LIN {X 0,Y 286.742,Z 491.523,A -85,B 0,C 180,E1 -18513.428,E2 -18513.428} C_VEL
LIN {X 0,Y 283.186,Z 502.115,A -85,B 0,C 180,E1 -18515.045,E2 -18515.045} C_VEL
LIN {X 0,Y 279.87,Z 510.827,A -85,B 0,C 180,E1 -18516.702,E2 -18516.702} C_VEL
LIN {X 0,Y 276.057,Z 519.397,A -85,B 0,C 180,E1 -18518.728,E2 -18518.728} C_VEL
LIN {X 0,Y 272.636,Z 526.32,A -85,B 0,C 180,E1 -18520.811,E2 -18520.811} C_VEL
LIN {X 0,Y 269.962,Z 531.061,A -85,B 0,C 180,E1 -18522.579,E2 -18522.579} C_VEL
LIN {X 0,Y 267.064,Z 535.632,A -85,B 0,C 180,E1 -18524.742,E2 -18524.742} C_VEL
LIN {X 0,Y 265.332,Z 538.078,A -85,B 0,C 180,E1 -18526.208,E2 -18526.208} C_VEL
LIN {X 0,Y 263.694,Z 540.035,A -85,B 0,C 180,E1 -18527.688,E2 -18527.688} C_VEL
LIN {X 0,Y 262.269,Z 541.552,A -85,B 0,C 180,E1 -18529.188,E2 -18529.188} C_VEL
LIN {X 0,Y 260.929,Z 542.67,A -85,B 0,C 180,E1 -18530.699,E2 -18530.699} C_VEL
LIN {X 0,Y 259.796,Z 543.334,A -85,B 0,C 180,E1 -18532.226,E2 -18532.226} C_VEL
LIN {X 0,Y 257.917,Z 543.43,A -85,B 0,C 180,E1 -18535.31,E2 -18535.31} C_VEL
LIN {X 0,Y 257.232,Z 542.868,A -85,B 0,C 180,E1 -18536.867,E2 -18536.867} C_VEL
LIN {X 0,Y 256.673,Z 541.852,A -85,B 0,C 180,E1 -18538.43,E2 -18538.43} C_VEL
LIN {X 0,Y 256.227,Z 540.428,A -85,B 0,C 180,E1 -18539.999,E2 -18539.999} C_VEL
LIN {X 0,Y 255.594,Z 537.491,A -85,B 0,C 180,E1 -18542.363,E2 -18542.363} C_VEL
LIN {X 0,Y 255.538,Z 533.499,A -85,B 0,C 180,E1 -18544.732,E2 -18544.732} C_VEL
LIN {X 0,Y 255.707,Z 527.917,A -85,B 0,C 180,E1 -18547.289,E2 -18547.289} C_VEL
LIN {X 0,Y 256.033,Z 520.721,A -85,B 0,C 180,E1 -18549.878,E2 -18549.878} C_VEL
LIN {X 0,Y 256.482,Z 512.466,A -85,B 0,C 180,E1 -18552.26,E2 -18552.26} C_VEL
LIN {X 0,Y 257.064,Z 504.113,A -85,B 0,C 180,E1 -18554.243,E2 -18554.243} C_VEL
LIN {X 0,Y 257.823,Z 493.991,A -85,B 0,C 180,E1 -18556.224,E2 -18556.224} C_VEL
LIN {X 0,Y 258.627,Z 482.98,A -85,B 0,C 180,E1 -18557.991,E2 -18557.991} C_VEL
LIN {X 0,Y 259.558,Z 470.695,A -85,B 0,C 180,E1 -18559.576,E2 -18559.576} C_VEL
LIN {X 0,Y 260.256,Z 456.947,A -85,B 0,C 180,E1 -18560.965,E2 -18560.965} C_VEL
LIN {X 0,Y 260.958,Z 443.101,A -85,B 0,C 180,E1 -18561.994,E2 -18561.994} C_VEL
LIN {X 0,Y 261.321,Z 428.706,A -85,B 0,C 180,E1 -18562.742,E2 -18562.742} C_VEL
LIN {X 0,Y 263.063,Z 376.798,A -85,B 0,C 180,E1 -18564.915,E2 -18564.915} C_VEL
LIN {X 0,Y 263.115,Z 373.058,A -85,B 0,C 180,E1 -18565.074,E2 -18565.074} C_VEL
LIN {X 0,Y 256.217,Z 349.569,A -85,B 0,C 180,E1 -18566.43,E2 -18566.43} C_VEL
LIN {X 0,Y 256.113,Z 349.578,A -85,B 0,C 180,E1 -18569.599,E2 -18569.599} C_VEL
LIN {X 0,Y 256.067,Z 349.587,A -85,B 0,C 180,E1 -18573.292,E2 -18573.292} C_VEL
LIN {X 0,Y 256.112,Z 349.58,A -85,B 0,C 180,E1 -18577.27,E2 -18577.27} C_VEL
LIN {X 0,Y 256.053,Z 349.589,A -85,B 0,C 180,E1 -18581.203,E2 -18581.203} C_VEL
LIN {X 0,Y 256.06,Z 349.586,A -85,B 0,C 180,E1 -18585.529,E2 -18585.529} C_VEL
LIN {X 0,Y 256.055,Z 349.591,A -85,B 0,C 180,E1 -18588.797,E2 -18588.797} C_VEL
LIN {X 0,Y 256.143,Z 349.579,A -85,B 0,C 180,E1 -18592.87,E2 -18592.87} C_VEL
LIN {X 0,Y 256.082,Z 349.587,A -85,B 0,C 180,E1 -18596.709,E2 -18596.709} C_VEL
LIN {X 0,Y 256.124,Z 349.579,A -85,B 0,C 180,E1 -18601.409,E2 -18601.409} C_VEL
LIN {X 0,Y 256.164,Z 349.573,A -85,B 0,C 180,E1 -18605.699,E2 -18605.699} C_VEL
LIN {X 0,Y 256.165,Z 349.574,A -85,B 0,C 180,E1 -18609.105,E2 -18609.105} C_VEL
LIN {X 0,Y 256.297,Z 349.557,A -85,B 0,C 180,E1 -18614.085,E2 -18614.085} C_VEL
LIN {X 0,Y 256.307,Z 349.556,A -85,B 0,C 180,E1 -18618.934,E2 -18618.934} C_VEL
LIN {X 0,Y 256.538,Z 349.527,A -85,B 0,C 180,E1 -18622.127,E2 -18622.127} C_VEL
LIN {X 0,Y 256.712,Z 349.508,A -85,B 0,C 180,E1 -18628.431,E2 -18628.431} C_VEL
LIN {X 0,Y 256.712,Z 349.505,A -85,B 0,C 180,E1 -18631.569,E2 -18631.569} C_VEL
LIN {X 0,Y 256.538,Z 349.527,A -85,B 0,C 180,E1 -18637.873,E2 -18637.873} C_VEL
LIN {X 0,Y 256.307,Z 349.556,A -85,B 0,C 180,E1 -18641.066,E2 -18641.066} C_VEL
LIN {X 0,Y 256.298,Z 349.558,A -85,B 0,C 180,E1 -18645.915,E2 -18645.915} C_VEL
LIN {X 0,Y 256.165,Z 349.574,A -85,B 0,C 180,E1 -18650.896,E2 -18650.896} C_VEL
LIN {X 0,Y 256.187,Z 349.569,A -85,B 0,C 180,E1 -18655.139,E2 -18655.139} C_VEL
LIN {X 0,Y 256.102,Z 349.582,A -85,B 0,C 180,E1 -18659.602,E2 -18659.602} C_VEL
LIN {X 0,Y 256.084,Z 349.582,A -85,B 0,C 180,E1 -18663.291,E2 -18663.291} C_VEL
LIN {X 0,Y 256.127,Z 349.578,A -85,B 0,C 180,E1 -18667.276,E2 -18667.276} C_VEL
LIN {X 0,Y 256.056,Z 349.586,A -85,B 0,C 180,E1 -18671.204,E2 -18671.204} C_VEL
LIN {X 0,Y 256.057,Z 349.588,A -85,B 0,C 180,E1 -18675.531,E2 -18675.531} C_VEL
LIN {X 0,Y 256.054,Z 349.587,A -85,B 0,C 180,E1 -18678.798,E2 -18678.798} C_VEL
LIN {X 0,Y 256.139,Z 349.576,A -85,B 0,C 180,E1 -18682.87,E2 -18682.87} C_VEL
LIN {X 0,Y 256.132,Z 349.577,A -85,B 0,C 180,E1 -18687.122,E2 -18687.122} C_VEL
LIN {X 0,Y 263.843,Z 373.942,A -85,B 0,C 180,E1 -18688.527,E2 -18688.527} C_VEL
LIN {X 0,Y 261.875,Z 433.631,A -85,B 0,C 180,E1 -18690.895,E2 -18690.895} C_VEL
LIN {X 0,Y 261.396,Z 447.781,A -85,B 0,C 180,E1 -18691.715,E2 -18691.715} C_VEL
LIN {X 0,Y 260.706,Z 461.252,A -85,B 0,C 180,E1 -18692.824,E2 -18692.824} C_VEL
LIN {X 0,Y 259.893,Z 473.611,A -85,B 0,C 180,E1 -18694.149,E2 -18694.149} C_VEL
LIN {X 0,Y 258.984,Z 485.469,A -85,B 0,C 180,E1 -18695.768,E2 -18695.768} C_VEL
LIN {X 0,Y 258.047,Z 496.288,A -85,B 0,C 180,E1 -18697.587,E2 -18697.587} C_VEL
LIN {X 0,Y 257.243,Z 506.028,A -85,B 0,C 180,E1 -18699.615,E2 -18699.615} C_VEL
LIN {X 0,Y 256.505,Z 515.525,A -85,B 0,C 180,E1 -18702.048,E2 -18702.048} C_VEL
LIN {X 0,Y 255.992,Z 523.081,A -85,B 0,C 180,E1 -18704.475,E2 -18704.475} C_VEL
LIN {X 0,Y 255.613,Z 530.03,A -85,B 0,C 180,E1 -18707.294,E2 -18707.294} C_VEL
LIN {X 0,Y 255.63,Z 534.568,A -85,B 0,C 180,E1 -18709.707,E2 -18709.707} C_VEL
LIN {X 0,Y 255.9,Z 537.977,A -85,B 0,C 180,E1 -18712.108,E2 -18712.108} C_VEL
LIN {X 0,Y 256.113,Z 539.674,A -85,B 0,C 180,E1 -18713.699,E2 -18713.699} C_VEL
LIN {X 0,Y 256.404,Z 540.938,A -85,B 0,C 180,E1 -18715.284,E2 -18715.284} C_VEL
LIN {X 0,Y 256.951,Z 541.725,A -85,B 0,C 180,E1 -18716.865,E2 -18716.865} C_VEL
LIN {X 0,Y 257.624,Z 542.11,A -85,B 0,C 180,E1 -18718.438,E2 -18718.438} C_VEL
LIN {X 0,Y 258.435,Z 542.082,A -85,B 0,C 180,E1 -18720.001,E2 -18720.001} C_VEL
LIN {X 0,Y 259.323,Z 541.593,A -85,B 0,C 180,E1 -18721.554,E2 -18721.554} C_VEL
LIN {X 0,Y 261.561,Z 539.402,A -85,B 0,C 180,E1 -18724.624,E2 -18724.624} C_VEL
LIN {X 0,Y 263.689,Z 536.578,A -85,B 0,C 180,E1 -18726.889,E2 -18726.889} C_VEL
LIN {X 0,Y 266.034,Z 532.7,A -85,B 0,C 180,E1 -18729.121,E2 -18729.121} C_VEL
LIN {X 0,Y 267.361,Z 530.257,A -85,B 0,C 180,E1 -18730.227,E2 -18730.227} C_VEL
LIN {X 0,Y 268.185,Z 527.805,A -85,B 0,C 180,E1 -18731.362,E2 -18731.362} C_VEL
LIN {X 0,Y 268.143,Z 523.856,A -85,B 0,C 180,E1 -18733.306,E2 -18733.306} C_VEL
LIN {X 0,Y 268.21,Z 519.378,A -85,B 0,C 180,E1 -18735.187,E2 -18735.187} C_VEL
LIN {X 0,Y 269.162,Z 516.063,A -85,B 0,C 180,E1 -18736.204,E2 -18736.204} C_VEL
LIN {X 0,Y 272.495,Z 507.969,A -85,B 0,C 180,E1 -18738.03,E2 -18738.03} C_VEL
LIN {X 0,Y 275.746,Z 498.639,A -85,B 0,C 180,E1 -18739.738,E2 -18739.738} C_VEL
LIN {X 0,Y 279.246,Z 487.143,A -85,B 0,C 180,E1 -18741.405,E2 -18741.405} C_VEL
LIN {X 0,Y 282.117,Z 475.634,A -85,B 0,C 180,E1 -18742.715,E2 -18742.715} C_VEL
LIN {X 0,Y 284.548,Z 462.972,A -85,B 0,C 180,E1 -18743.857,E2 -18743.857} C_VEL
LIN {X 0,Y 286.529,Z 448.771,A -85,B 0,C 180,E1 -18744.817,E2 -18744.817} C_VEL
LIN {X 0,Y 289.784,Z 421.766,A -85,B 0,C 180,E1 -18746.079,E2 -18746.079} C_VEL
LIN {X 0,Y 291.826,Z 407.158,A -85,B 0,C 180,E1 -18746.682,E2 -18746.682} C_VEL
LIN {X 0,Y 288.803,Z 401.044,A -85,B 0,C 180,E1 -18748.509,E2 -18748.509} C_VEL
LIN {X 0,Y 286.95,Z 397.572,A -85,B 0,C 180,E1 -18749.809,E2 -18749.809} C_VEL
LIN {X 0,Y 285.256,Z 394.534,A -85,B 0,C 180,E1 -18751.158,E2 -18751.158} C_VEL
LIN {X 0,Y 283.356,Z 391.067,A -85,B 0,C 180,E1 -18753.009,E2 -18753.009} C_VEL
LIN {X 0,Y 281.225,Z 387.965,A -85,B 0,C 180,E1 -18755.844,E2 -18755.844} C_VEL
LIN {X 0,Y 280.356,Z 386.885,A -85,B 0,C 180,E1 -18757.914,E2 -18757.914} C_VEL
LIN {X 0,Y 279.977,Z 387.1,A -85,B 0,C 180,E1 -18760.122,E2 -18760.122} C_VEL
LIN {X 0,Y 280.903,Z 389.538,A -85,B 0,C 180,E1 -18763.905,E2 -18763.905} C_VEL
LIN {X 0,Y 281.598,Z 390.488,A -85,B 0,C 180,E1 -18764.946,E2 -18764.946} C_VEL
LIN {X 0,Y 284.076,Z 395.271,A -85,B 0,C 180,E1 -18767.92,E2 -18767.92} C_VEL
LIN {X 0,Y 285.9,Z 398.582,A -85,B 0,C 180,E1 -18769.468,E2 -18769.468} C_VEL
LIN {X 0,Y 287.386,Z 407.637,A -85,B 0,C 180,E1 -18771.281,E2 -18771.281} C_VEL
LIN {X 0,Y 287.167,Z 422.972,A -85,B 0,C 180,E1 -18772.78,E2 -18772.78} C_VEL
LIN {X 0,Y 286.547,Z 444.861,A -85,B 0,C 180,E1 -18774.577,E2 -18774.577} C_VEL
LIN {X 0,Y 285.739,Z 460.739,A -85,B 0,C 180,E1 -18775.664,E2 -18775.664} C_VEL
LIN {X 0,Y 281.973,Z 489.26,A -85,B 0,C 180,E1 -18776.906,E2 -18776.906} C_VEL
LIN {X 0,Y 279.037,Z 503.696,A -85,B 0,C 180,E1 -18777.748,E2 -18777.748} C_VEL
LIN {X 0,Y 275.393,Z 517.912,A -85,B 0,C 180,E1 -18778.883,E2 -18778.883} C_VEL
LIN {X 0,Y 271.17,Z 531.452,A -85,B 0,C 180,E1 -18780.286,E2 -18780.286} C_VEL
LIN {X 0,Y 266.886,Z 543.474,A -85,B 0,C 180,E1 -18781.919,E2 -18781.919} C_VEL
LIN {X 0,Y 262.716,Z 554.359,A -85,B 0,C 180,E1 -18783.807,E2 -18783.807} C_VEL
LIN {X 0,Y 258.893,Z 564.083,A -85,B 0,C 180,E1 -18785.971,E2 -18785.971} C_VEL
LIN {X 0,Y 254.961,Z 573.385,A -85,B 0,C 180,E1 -18788.577,E2 -18788.577} C_VEL
LIN {X 0,Y 252.27,Z 579.962,A -85,B 0,C 180,E1 -18790.934,E2 -18790.934} C_VEL
LIN {X 0,Y 250.077,Z 585.908,A -85,B 0,C 180,E1 -18793.678,E2 -18793.678} C_VEL
LIN {X 0,Y 248.683,Z 589.992,A -85,B 0,C 180,E1 -18796.1,E2 -18796.1} C_VEL
LIN {X 0,Y 247.839,Z 593.104,A -85,B 0,C 180,E1 -18798.55,E2 -18798.55} C_VEL
LIN {X 0,Y 247.57,Z 595.814,A -85,B 0,C 180,E1 -18801.84,E2 -18801.84} C_VEL
LIN {X 0,Y 247.782,Z 596.584,A -85,B 0,C 180,E1 -18803.485,E2 -18803.485} C_VEL
LIN {X 0,Y 248.084,Z 596.901,A -85,B 0,C 180,E1 -18805.124,E2 -18805.124} C_VEL
LIN {X 0,Y 248.393,Z 596.776,A -85,B 0,C 180,E1 -18806.756,E2 -18806.756} C_VEL
LIN {X 0,Y 249.218,Z 595.365,A -85,B 0,C 180,E1 -18809.798,E2 -18809.798} C_VEL
LIN {X 0,Y 248.814,Z 596.563,A -85,B 0,C 180,E1 -18811.618,E2 -18811.618} C_VEL
LIN {X 0,Y 248.404,Z 597.315,A -85,B 0,C 180,E1 -18813.244,E2 -18813.244} C_VEL
LIN {X 0,Y 248.06,Z 597.605,A -85,B 0,C 180,E1 -18814.876,E2 -18814.876} C_VEL
LIN {X 0,Y 247.726,Z 597.376,A -85,B 0,C 180,E1 -18816.801,E2 -18816.801} C_VEL
LIN {X 0,Y 247.558,Z 595.93,A -85,B 0,C 180,E1 -18819.807,E2 -18819.807} C_VEL
LIN {X 0,Y 248.302,Z 592.866,A -85,B 0,C 180,E1 -18823.087,E2 -18823.087} C_VEL
LIN {X 0,Y 250.092,Z 588.158,A -85,B 0,C 180,E1 -18826.321,E2 -18826.321} C_VEL
LIN {X 0,Y 251.999,Z 583.525,A -85,B 0,C 180,E1 -18828.706,E2 -18828.706} C_VEL
LIN {X 0,Y 255.059,Z 576.787,A -85,B 0,C 180,E1 -18831.413,E2 -18831.413} C_VEL
LIN {X 0,Y 258.962,Z 568.425,A -85,B 0,C 180,E1 -18834.022,E2 -18834.022} C_VEL
LIN {X 0,Y 263.68,Z 558.098,A -85,B 0,C 180,E1 -18836.516,E2 -18836.516} C_VEL
LIN {X 0,Y 268.353,Z 547.299,A -85,B 0,C 180,E1 -18838.552,E2 -18838.552} C_VEL
LIN {X 0,Y 273.264,Z 535.286,A -85,B 0,C 180,E1 -18840.313,E2 -18840.313} C_VEL
LIN {X 0,Y 278.14,Z 521.862,A -85,B 0,C 180,E1 -18841.834,E2 -18841.834} C_VEL
LIN {X 0,Y 281.737,Z 510.521,A -85,B 0,C 180,E1 -18842.858,E2 -18842.858} C_VEL
LIN {X 0,Y 285.669,Z 496.262,A -85,B 0,C 180,E1 -18843.822,E2 -18843.822} C_VEL
LIN {X 0,Y 288.719,Z 481.403,A -85,B 0,C 180,E1 -18844.627,E2 -18844.627} C_VEL
LIN {X 0,Y 291.912,Z 460.369,A -85,B 0,C 180,E1 -18845.6,E2 -18845.6} C_VEL
LIN {X 0,Y 292.903,Z 448.794,A -85,B 0,C 180,E1 -18846.446,E2 -18846.446} C_VEL
LIN {X 0,Y 293.578,Z 434.493,A -85,B 0,C 180,E1 -18847.843,E2 -18847.843} C_VEL
LIN {X 0,Y 293.851,Z 424.317,A -85,B 0,C 180,E1 -18849.08,E2 -18849.08} C_VEL
LIN {X 0,Y 292.771,Z 419.312,A -85,B 0,C 180,E1 -18850.545,E2 -18850.545} C_VEL
LIN {X 0,Y 291.269,Z 412.435,A -85,B 0,C 180,E1 -18853.385,E2 -18853.385} C_VEL
LIN {X 0,Y 290.688,Z 408.854,A -85,B 0,C 180,E1 -18855.965,E2 -18855.965} C_VEL
LIN {X 0,Y 291.094,Z 406.843,A -85,B 0,C 180,E1 -18858.456,E2 -18858.456} C_VEL
LIN {X 0,Y 291.913,Z 406.771,A -85,B 0,C 180,E1 -18860.392,E2 -18860.392} C_VEL
LIN {X 0,Y 293.782,Z 407.401,A -85,B 0,C 180,E1 -18862.724,E2 -18862.724} C_VEL
LIN {X 0,Y 295.754,Z 409.575,A -85,B 0,C 180,E1 -18864.604,E2 -18864.604} C_VEL
LIN {X 0,Y 298.261,Z 412.85,A -85,B 0,C 180,E1 -18866.477,E2 -18866.477} C_VEL
LIN {X 0,Y 297.816,Z 415.868,A -85,B 0,C 180,E1 -18866.654,E2 -18866.654} C_VEL
LIN {X 0,Y 293.769,Z 440.311,A -85,B 0,C 180,E1 -18867.795,E2 -18867.795} C_VEL
LIN {X 0,Y 291.149,Z 457.751,A -85,B 0,C 180,E1 -18868.786,E2 -18868.786} C_VEL
LIN {X 0,Y 288.547,Z 471.053,A -85,B 0,C 180,E1 -18869.843,E2 -18869.843} C_VEL
LIN {X 0,Y 285.415,Z 483.408,A -85,B 0,C 180,E1 -18871.102,E2 -18871.102} C_VEL
LIN {X 0,Y 281.946,Z 494.551,A -85,B 0,C 180,E1 -18872.538,E2 -18872.538} C_VEL
LIN {X 0,Y 278.186,Z 504.776,A -85,B 0,C 180,E1 -18874.163,E2 -18874.163} C_VEL
LIN {X 0,Y 273.943,Z 514.669,A -85,B 0,C 180,E1 -18876.167,E2 -18876.167} C_VEL
LIN {X 0,Y 270,Z 522.712,A -85,B 0,C 180,E1 -18878.227,E2 -18878.227} C_VEL
LIN {X 0,Y 265.813,Z 530.132,A -85,B 0,C 180,E1 -18880.7,E2 -18880.7} C_VEL
LIN {X 0,Y 262.542,Z 535.137,A -85,B 0,C 180,E1 -18882.874,E2 -18882.874} C_VEL
LIN {X 0,Y 259.618,Z 539.02,A -85,B 0,C 180,E1 -18885.097,E2 -18885.097} C_VEL
LIN {X 0,Y 256.985,Z 541.867,A -85,B 0,C 180,E1 -18887.362,E2 -18887.362} C_VEL
LIN {X 0,Y 255.485,Z 543.207,A -85,B 0,C 180,E1 -18888.897,E2 -18888.897} C_VEL
LIN {X 0,Y 254.087,Z 544.115,A -85,B 0,C 180,E1 -18890.446,E2 -18890.446} C_VEL
LIN {X 0,Y 251.849,Z 544.726,A -85,B 0,C 180,E1 -18893.59,E2 -18893.59} C_VEL
LIN {X 0,Y 250.93,Z 544.402,A -85,B 0,C 180,E1 -18895.179,E2 -18895.179} C_VEL
LIN {X 0,Y 249.623,Z 542.495,A -85,B 0,C 180,E1 -18898.386,E2 -18898.386} C_VEL
LIN {X 0,Y 248.874,Z 539.968,A -85,B 0,C 180,E1 -18900.808,E2 -18900.808} C_VEL
LIN {X 0,Y 248.416,Z 536.436,A -85,B 0,C 180,E1 -18903.243,E2 -18903.243} C_VEL
LIN {X 0,Y 248.531,Z 531.809,A -85,B 0,C 180,E1 -18905.679,E2 -18905.679} C_VEL
LIN {X 0,Y 248.705,Z 524.98,A -85,B 0,C 180,E1 -18908.49,E2 -18908.49} C_VEL
LIN {X 0,Y 249.127,Z 517.349,A -85,B 0,C 180,E1 -18910.977,E2 -18910.977} C_VEL
LIN {X 0,Y 249.714,Z 508.079,A -85,B 0,C 180,E1 -18913.425,E2 -18913.425} C_VEL
LIN {X 0,Y 250.556,Z 497.595,A -85,B 0,C 180,E1 -18915.662,E2 -18915.662} C_VEL
LIN {X 0,Y 251.245,Z 487.082,A -85,B 0,C 180,E1 -18917.499,E2 -18917.499} C_VEL
LIN {X 0,Y 252.224,Z 474.131,A -85,B 0,C 180,E1 -18919.31,E2 -18919.31} C_VEL
LIN {X 0,Y 253.016,Z 461.087,A -85,B 0,C 180,E1 -18920.741,E2 -18920.741} C_VEL
LIN {X 0,Y 253.726,Z 447.858,A -85,B 0,C 180,E1 -18921.851,E2 -18921.851} C_VEL
LIN {X 0,Y 254.156,Z 434.342,A -85,B 0,C 180,E1 -18922.668,E2 -18922.668} C_VEL
LIN {X 0,Y 255.896,Z 380.734,A -85,B 0,C 180,E1 -18925.014,E2 -18925.014} C_VEL
LIN {X 0,Y 256.129,Z 374.232,A -85,B 0,C 180,E1 -18925.297,E2 -18925.297} C_VEL
LIN {X 0,Y 249.179,Z 350.447,A -85,B 0,C 180,E1 -18926.69,E2 -18926.69} C_VEL
LIN {X 0,Y 249.051,Z 350.459,A -85,B 0,C 180,E1 -18930.526,E2 -18930.526} C_VEL
LIN {X 0,Y 249.043,Z 350.463,A -85,B 0,C 180,E1 -18935.077,E2 -18935.077} C_VEL
LIN {X 0,Y 249.024,Z 350.463,A -85,B 0,C 180,E1 -18938.38,E2 -18938.38} C_VEL
LIN {X 0,Y 249.01,Z 350.469,A -85,B 0,C 180,E1 -18942.793,E2 -18942.793} C_VEL
LIN {X 0,Y 249.016,Z 350.463,A -85,B 0,C 180,E1 -18947.363,E2 -18947.363} C_VEL
LIN {X 0,Y 249.036,Z 350.462,A -85,B 0,C 180,E1 -18951.621,E2 -18951.621} C_VEL
LIN {X 0,Y 249.059,Z 350.456,A -85,B 0,C 180,E1 -18955.642,E2 -18955.642} C_VEL
LIN {X 0,Y 249.045,Z 350.461,A -85,B 0,C 180,E1 -18959.472,E2 -18959.472} C_VEL
LIN {X 0,Y 249.069,Z 350.456,A -85,B 0,C 180,E1 -18963.162,E2 -18963.162} C_VEL
LIN {X 0,Y 249.077,Z 350.46,A -85,B 0,C 180,E1 -18966.733,E2 -18966.733} C_VEL
LIN {X 0,Y 249.108,Z 350.455,A -85,B 0,C 180,E1 -18970.212,E2 -18970.212} C_VEL
LIN {X 0,Y 249.239,Z 350.435,A -85,B 0,C 180,E1 -18973.622,E2 -18973.622} C_VEL
LIN {X 0,Y 249.25,Z 350.438,A -85,B 0,C 180,E1 -18978.617,E2 -18978.617} C_VEL
LIN {X 0,Y 249.482,Z 350.405,A -85,B 0,C 180,E1 -18981.903,E2 -18981.903} C_VEL
LIN {X 0,Y 249.435,Z 350.413,A -85,B 0,C 180,E1 -18986.77,E2 -18986.77} C_VEL
LIN {X 0,Y 249.726,Z 350.375,A -85,B 0,C 180,E1 -18990,E2 -18990} C_VEL
LIN {X 0,Y 249.435,Z 350.412,A -85,B 0,C 180,E1 -18993.231,E2 -18993.231} C_VEL
LIN {X 0,Y 249.482,Z 350.407,A -85,B 0,C 180,E1 -18998.097,E2 -18998.097} C_VEL
LIN {X 0,Y 249.251,Z 350.435,A -85,B 0,C 180,E1 -19001.384,E2 -19001.384} C_VEL
LIN {X 0,Y 249.24,Z 350.437,A -85,B 0,C 180,E1 -19006.379,E2 -19006.379} C_VEL
LIN {X 0,Y 249.085,Z 350.456,A -85,B 0,C 180,E1 -19011.519,E2 -19011.519} C_VEL
LIN {X 0,Y 249.129,Z 350.448,A -85,B 0,C 180,E1 -19015.483,E2 -19015.483} C_VEL
LIN {X 0,Y 249.072,Z 350.457,A -85,B 0,C 180,E1 -19018.99,E2 -19018.99} C_VEL
LIN {X 0,Y 249.035,Z 350.463,A -85,B 0,C 180,E1 -19022.426,E2 -19022.426} C_VEL
LIN {X 0,Y 249.068,Z 350.46,A -85,B 0,C 180,E1 -19026.34,E2 -19026.34} C_VEL
LIN {X 0,Y 249.025,Z 350.464,A -85,B 0,C 180,E1 -19030.475,E2 -19030.475} C_VEL
LIN {X 0,Y 249.002,Z 350.466,A -85,B 0,C 180,E1 -19034.88,E2 -19034.88} C_VEL
LIN {X 0,Y 249.016,Z 350.465,A -85,B 0,C 180,E1 -19037.364,E2 -19037.364} C_VEL
LIN {X 0,Y 249.049,Z 350.462,A -85,B 0,C 180,E1 -19042.2,E2 -19042.2} C_VEL
LIN {X 0,Y 249.092,Z 350.478,A -85,B 0,C 180,E1 -19046.79,E2 -19046.79} C_VEL
LIN {X 0,Y 256.898,Z 375.833,A -85,B 0,C 180,E1 -19048.285,E2 -19048.285} C_VEL
LIN {X 0,Y 254.883,Z 432.986,A -85,B 0,C 180,E1 -19050.613,E2 -19050.613} C_VEL
LIN {X 0,Y 254.434,Z 447.193,A -85,B 0,C 180,E1 -19051.432,E2 -19051.432} C_VEL
LIN {X 0,Y 253.763,Z 460.036,A -85,B 0,C 180,E1 -19052.476,E2 -19052.476} C_VEL
LIN {X 0,Y 252.937,Z 472.635,A -85,B 0,C 180,E1 -19053.827,E2 -19053.827} C_VEL
LIN {X 0,Y 252.004,Z 484.871,A -85,B 0,C 180,E1 -19055.492,E2 -19055.492} C_VEL
LIN {X 0,Y 250.951,Z 496.891,A -85,B 0,C 180,E1 -19057.547,E2 -19057.547} C_VEL
LIN {X 0,Y 250.184,Z 505.895,A -85,B 0,C 180,E1 -19059.444,E2 -19059.444} C_VEL
LIN {X 0,Y 249.439,Z 515.614,A -85,B 0,C 180,E1 -19061.946,E2 -19061.946} C_VEL
LIN {X 0,Y 248.919,Z 523.407,A -85,B 0,C 180,E1 -19064.457,E2 -19064.457} C_VEL
LIN {X 0,Y 248.551,Z 529.577,A -85,B 0,C 180,E1 -19066.927,E2 -19066.927} C_VEL
LIN {X 0,Y 248.553,Z 534.468,A -85,B 0,C 180,E1 -19069.41,E2 -19069.41} C_VEL
LIN {X 0,Y 248.797,Z 538.174,A -85,B 0,C 180,E1 -19071.881,E2 -19071.881} C_VEL
LIN {X 0,Y 249.016,Z 540.05,A -85,B 0,C 180,E1 -19073.519,E2 -19073.519} C_VEL
LIN {X 0,Y 249.307,Z 541.478,A -85,B 0,C 180,E1 -19075.149,E2 -19075.149} C_VEL
LIN {X 0,Y 249.871,Z 542.496,A -85,B 0,C 180,E1 -19076.776,E2 -19076.776} C_VEL
LIN {X 0,Y 250.548,Z 543.064,A -85,B 0,C 180,E1 -19078.393,E2 -19078.393} C_VEL
LIN {X 0,Y 252.307,Z 542.923,A -85,B 0,C 180,E1 -19081.597,E2 -19081.597} C_VEL
LIN {X 0,Y 253.445,Z 542.235,A -85,B 0,C 180,E1 -19083.18,E2 -19083.18} C_VEL
LIN {X 0,Y 254.627,Z 541.104,A -85,B 0,C 180,E1 -19084.75,E2 -19084.75} C_VEL
LIN {X 0,Y 256.846,Z 538.57,A -85,B 0,C 180,E1 -19087.074,E2 -19087.074} C_VEL
LIN {X 0,Y 259.285,Z 535.044,A -85,B 0,C 180,E1 -19089.36,E2 -19089.36} C_VEL
LIN {X 0,Y 262.125,Z 530.385,A -85,B 0,C 180,E1 -19091.601,E2 -19091.601} C_VEL
LIN {X 0,Y 265.284,Z 524.457,A -85,B 0,C 180,E1 -19093.795,E2 -19093.795} C_VEL
LIN {X 0,Y 269.162,Z 516.063,A -85,B 0,C 180,E1 -19096.204,E2 -19096.204} C_VEL
LIN {X 0,Y 270.174,Z 512.554,A -85,B 0,C 180,E1 -19097.195,E2 -19097.195} C_VEL
LIN {X 0,Y 270.594,Z 506.948,A -85,B 0,C 180,E1 -19098.929,E2 -19098.929} C_VEL
LIN {X 0,Y 271.129,Z 500.895,A -85,B 0,C 180,E1 -19100.562,E2 -19100.562} C_VEL
LIN {X 0,Y 272.258,Z 496.597,A -85,B 0,C 180,E1 -19101.379,E2 -19101.379} C_VEL
LIN {X 0,Y 275.998,Z 484.252,A -85,B 0,C 180,E1 -19103.049,E2 -19103.049} C_VEL
LIN {X 0,Y 279.032,Z 471.916,A -85,B 0,C 180,E1 -19104.359,E2 -19104.359} C_VEL
LIN {X 0,Y 281.266,Z 460.165,A -85,B 0,C 180,E1 -19105.335,E2 -19105.335} C_VEL
LIN {X 0,Y 283.058,Z 446.969,A -85,B 0,C 180,E1 -19106.15,E2 -19106.15} C_VEL
LIN {X 0,Y 286.825,Z 419.106,A -85,B 0,C 180,E1 -19107.444,E2 -19107.444} C_VEL
LIN {X 0,Y 288.004,Z 410.935,A -85,B 0,C 180,E1 -19107.809,E2 -19107.809} C_VEL
LIN {X 0,Y 285.543,Z 405.838,A -85,B 0,C 180,E1 -19109.49,E2 -19109.49} C_VEL
LIN {X 0,Y 283.131,Z 401.134,A -85,B 0,C 180,E1 -19111.47,E2 -19111.47} C_VEL
LIN {X 0,Y 281.086,Z 397.38,A -85,B 0,C 180,E1 -19113.626,E2 -19113.626} C_VEL
LIN {X 0,Y 279.194,Z 394.309,A -85,B 0,C 180,E1 -19116.68,E2 -19116.68} C_VEL
LIN {X 0,Y 278.57,Z 393.765,A -85,B 0,C 180,E1 -19118.546,E2 -19118.546} C_VEL
LIN {X 0,Y 278.353,Z 394.166,A -85,B 0,C 180,E1 -19120.405,E2 -19120.405} C_VEL
LIN {X 0,Y 279.461,Z 396.637,A -85,B 0,C 180,E1 -19124.2,E2 -19124.2} C_VEL
LIN {X 0,Y 281.881,Z 401.602,A -85,B 0,C 180,E1 -19127.454,E2 -19127.454} C_VEL
LIN {X 0,Y 283.302,Z 404.465,A -85,B 0,C 180,E1 -19128.798,E2 -19128.798} C_VEL
LIN {X 0,Y 284.249,Z 411.59,A -85,B 0,C 180,E1 -19130.266,E2 -19130.266} C_VEL
LIN {X 0,Y 283.542,Z 429.178,A -85,B 0,C 180,E1 -19131.969,E2 -19131.969} C_VEL
LIN {X 0,Y 282.641,Z 448.887,A -85,B 0,C 180,E1 -19133.594,E2 -19133.594} C_VEL
LIN {X 0,Y 281.646,Z 463.52,A -85,B 0,C 180,E1 -19134.575,E2 -19134.575} C_VEL
LIN {X 0,Y 278.048,Z 488.271,A -85,B 0,C 180,E1 -19135.668,E2 -19135.668} C_VEL
LIN {X 0,Y 274.852,Z 502.906,A -85,B 0,C 180,E1 -19136.539,E2 -19136.539} C_VEL
LIN {X 0,Y 271.017,Z 517.025,A -85,B 0,C 180,E1 -19137.666,E2 -19137.666} C_VEL
LIN {X 0,Y 266.569,Z 530.354,A -85,B 0,C 180,E1 -19139.061,E2 -19139.061} C_VEL
LIN {X 0,Y 261.594,Z 543.36,A -85,B 0,C 180,E1 -19140.859,E2 -19140.859} C_VEL
LIN {X 0,Y 257.194,Z 554.004,A -85,B 0,C 180,E1 -19142.76,E2 -19142.76} C_VEL
LIN {X 0,Y 253.13,Z 563.494,A -85,B 0,C 180,E1 -19144.95,E2 -19144.95} C_VEL
LIN {X 0,Y 249.448,Z 571.48,A -85,B 0,C 180,E1 -19147.207,E2 -19147.207} C_VEL
LIN {X 0,Y 245.994,Z 579.008,A -85,B 0,C 180,E1 -19149.95,E2 -19149.95} C_VEL
LIN {X 0,Y 243.679,Z 584.659,A -85,B 0,C 180,E1 -19152.613,E2 -19152.613} C_VEL
LIN {X 0,Y 241.733,Z 589.583,A -85,B 0,C 180,E1 -19155.692,E2 -19155.692} C_VEL
LIN {X 0,Y 240.819,Z 592.487,A -85,B 0,C 180,E1 -19158.212,E2 -19158.212} C_VEL
LIN {X 0,Y 240.556,Z 593.942,A -85,B 0,C 180,E1 -19159.904,E2 -19159.904} C_VEL
LIN {X 0,Y 240.687,Z 595.568,A -85,B 0,C 180,E1 -19163.122,E2 -19163.122} C_VEL
LIN {X 0,Y 241.02,Z 595.819,A -85,B 0,C 180,E1 -19164.981,E2 -19164.981} C_VEL
LIN {X 0,Y 241.358,Z 595.609,A -85,B 0,C 180,E1 -19166.661,E2 -19166.661} C_VEL
LIN {X 0,Y 242.189,Z 594.188,A -85,B 0,C 180,E1 -19169.584,E2 -19169.584} C_VEL
LIN {X 0,Y 242.31,Z 593.862,A -85,B 0,C 180,E1 -19170,E2 -19170} C_VEL
LIN {X 0,Y 241.839,Z 595.147,A -85,B 0,C 180,E1 -19171.665,E2 -19171.665} C_VEL
LIN {X 0,Y 241.399,Z 595.983,A -85,B 0,C 180,E1 -19173.338,E2 -19173.338} C_VEL
LIN {X 0,Y 241.036,Z 596.394,A -85,B 0,C 180,E1 -19175.018,E2 -19175.018} C_VEL
LIN {X 0,Y 240.687,Z 596.361,A -85,B 0,C 180,E1 -19176.878,E2 -19176.878} C_VEL
LIN {X 0,Y 240.521,Z 595.104,A -85,B 0,C 180,E1 -19180.097,E2 -19180.097} C_VEL
LIN {X 0,Y 241.356,Z 592.294,A -85,B 0,C 180,E1 -19183.471,E2 -19183.471} C_VEL
LIN {X 0,Y 242.644,Z 589.168,A -85,B 0,C 180,E1 -19185.971,E2 -19185.971} C_VEL
LIN {X 0,Y 245.281,Z 583.578,A -85,B 0,C 180,E1 -19189.238,E2 -19189.238} C_VEL
LIN {X 0,Y 248.495,Z 577.205,A -85,B 0,C 180,E1 -19192.008,E2 -19192.008} C_VEL
LIN {X 0,Y 252.555,Z 569.265,A -85,B 0,C 180,E1 -19194.671,E2 -19194.671} C_VEL
LIN {X 0,Y 257.448,Z 559.543,A -85,B 0,C 180,E1 -19197.21,E2 -19197.21} C_VEL
LIN {X 0,Y 262.281,Z 549.376,A -85,B 0,C 180,E1 -19199.276,E2 -19199.276} C_VEL
LIN {X 0,Y 267.321,Z 538.19,A -85,B 0,C 180,E1 -19201.061,E2 -19201.061} C_VEL
LIN {X 0,Y 272.826,Z 524.496,A -85,B 0,C 180,E1 -19202.749,E2 -19202.749} C_VEL
LIN {X 0,Y 277.08,Z 512.363,A -85,B 0,C 180,E1 -19203.919,E2 -19203.919} C_VEL
LIN {X 0,Y 281.771,Z 497.013,A -85,B 0,C 180,E1 -19205.007,E2 -19205.007} C_VEL
LIN {X 0,Y 285.112,Z 482.358,A -85,B 0,C 180,E1 -19205.834,E2 -19205.834} C_VEL
LIN {X 0,Y 288.582,Z 461.513,A -85,B 0,C 180,E1 -19206.813,E2 -19206.813} C_VEL
LIN {X 0,Y 289.832,Z 448.835,A -85,B 0,C 180,E1 -19207.798,E2 -19207.798} C_VEL
LIN {X 0,Y 290.797,Z 434.472,A -85,B 0,C 180,E1 -19209.303,E2 -19209.303} C_VEL
LIN {X 0,Y 291.034,Z 429.012,A -85,B 0,C 180,E1 -19210.017,E2 -19210.017} C_VEL
LIN {X 0,Y 290.289,Z 424.939,A -85,B 0,C 180,E1 -19211.281,E2 -19211.281} C_VEL
LIN {X 0,Y 289.265,Z 418.908,A -85,B 0,C 180,E1 -19213.801,E2 -19213.801} C_VEL
LIN {X 0,Y 288.899,Z 415.656,A -85,B 0,C 180,E1 -19216.154,E2 -19216.154} C_VEL
LIN {X 0,Y 289.362,Z 413.71,A -85,B 0,C 180,E1 -19218.573,E2 -19218.573} C_VEL
LIN {X 0,Y 291.238,Z 413.94,A -85,B 0,C 180,E1 -19221.905,E2 -19221.905} C_VEL
LIN {X 0,Y 292.15,Z 414.603,A -85,B 0,C 180,E1 -19222.933,E2 -19222.933} C_VEL
LIN {X 0,Y 293.727,Z 416.368,A -85,B 0,C 180,E1 -19224.441,E2 -19224.441} C_VEL
LIN {X 0,Y 294.945,Z 417.973,A -85,B 0,C 180,E1 -19225.444,E2 -19225.444} C_VEL
LIN {X 0,Y 290.74,Z 441.673,A -85,B 0,C 180,E1 -19226.565,E2 -19226.565} C_VEL
LIN {X 0,Y 288.085,Z 458.048,A -85,B 0,C 180,E1 -19227.502,E2 -19227.502} C_VEL
LIN {X 0,Y 285.522,Z 470.485,A -85,B 0,C 180,E1 -19228.462,E2 -19228.462} C_VEL
LIN {X 0,Y 282.197,Z 483.034,A -85,B 0,C 180,E1 -19229.713,E2 -19229.713} C_VEL
LIN {X 0,Y 278.888,Z 493.289,A -85,B 0,C 180,E1 -19230.98,E2 -19230.98} C_VEL
LIN {X 0,Y 274.833,Z 503.826,A -85,B 0,C 180,E1 -19232.593,E2 -19232.593} C_VEL
LIN {X 0,Y 271.008,Z 512.515,A -85,B 0,C 180,E1 -19234.254,E2 -19234.254} C_VEL
LIN {X 0,Y 267.378,Z 519.822,A -85,B 0,C 180,E1 -19235.957,E2 -19235.957} C_VEL
LIN {X 0,Y 263.294,Z 527.076,A -85,B 0,C 180,E1 -19238.056,E2 -19238.056} C_VEL
LIN {X 0,Y 259.546,Z 532.9,A -85,B 0,C 180,E1 -19240.215,E2 -19240.215} C_VEL
LIN {X 0,Y 256.123,Z 537.528,A -85,B 0,C 180,E1 -19242.431,E2 -19242.431} C_VEL
LIN {X 0,Y 253.048,Z 541.081,A -85,B 0,C 180,E1 -19244.701,E2 -19244.701} C_VEL
LIN {X 0,Y 250.292,Z 543.638,A -85,B 0,C 180,E1 -19247.018,E2 -19247.018} C_VEL
LIN {X 0,Y 247.237,Z 545.551,A -85,B 0,C 180,E1 -19250.179,E2 -19250.179} C_VEL
LIN {X 0,Y 245.999,Z 545.877,A -85,B 0,C 180,E1 -19251.787,E2 -19251.787} C_VEL
LIN {X 0,Y 243.921,Z 545.296,A -85,B 0,C 180,E1 -19255.041,E2 -19255.041} C_VEL
LIN {X 0,Y 243.161,Z 544.406,A -85,B 0,C 180,E1 -19256.685,E2 -19256.685} C_VEL
LIN {X 0,Y 242.546,Z 543.076,A -85,B 0,C 180,E1 -19258.339,E2 -19258.339} C_VEL
LIN {X 0,Y 241.767,Z 540.301,A -85,B 0,C 180,E1 -19260.832,E2 -19260.832} C_VEL
LIN {X 0,Y 241.321,Z 536.502,A -85,B 0,C 180,E1 -19263.338,E2 -19263.338} C_VEL
LIN {X 0,Y 241.459,Z 531.592,A -85,B 0,C 180,E1 -19265.846,E2 -19265.846} C_VEL
LIN {X 0,Y 241.626,Z 524.967,A -85,B 0,C 180,E1 -19268.532,E2 -19268.532} C_VEL
LIN {X 0,Y 242,Z 517.826,A -85,B 0,C 180,E1 -19270.88,E2 -19270.88} C_VEL
LIN {X 0,Y 242.619,Z 508.435,A -85,B 0,C 180,E1 -19273.399,E2 -19273.399} C_VEL
LIN {X 0,Y 243.455,Z 497.838,A -85,B 0,C 180,E1 -19275.701,E2 -19275.701} C_VEL
LIN {X 0,Y 244.184,Z 487.146,A -85,B 0,C 180,E1 -19277.589,E2 -19277.589} C_VEL
LIN {X 0,Y 245.118,Z 474.443,A -85,B 0,C 180,E1 -19279.404,E2 -19279.404} C_VEL
LIN {X 0,Y 245.923,Z 461.829,A -85,B 0,C 180,E1 -19280.819,E2 -19280.819} C_VEL
LIN {X 0,Y 246.644,Z 448.656,A -85,B 0,C 180,E1 -19281.961,E2 -19281.961} C_VEL
LIN {X 0,Y 247.117,Z 434.103,A -85,B 0,C 180,E1 -19282.853,E2 -19282.853} C_VEL
LIN {X 0,Y 248.946,Z 379.997,A -85,B 0,C 180,E1 -19285.311,E2 -19285.311} C_VEL
LIN {X 0,Y 249.045,Z 375.114,A -85,B 0,C 180,E1 -19285.536,E2 -19285.536} C_VEL
LIN {X 0,Y 242.102,Z 351.328,A -85,B 0,C 180,E1 -19286.977,E2 -19286.977} C_VEL
LIN {X 0,Y 241.974,Z 351.341,A -85,B 0,C 180,E1 -19291.519,E2 -19291.519} C_VEL
LIN {X 0,Y 242.004,Z 351.337,A -85,B 0,C 180,E1 -19295.596,E2 -19295.596} C_VEL
LIN {X 0,Y 241.955,Z 351.342,A -85,B 0,C 180,E1 -19299.718,E2 -19299.718} C_VEL
LIN {X 0,Y 241.932,Z 351.347,A -85,B 0,C 180,E1 -19304.201,E2 -19304.201} C_VEL
LIN {X 0,Y 241.942,Z 351.344,A -85,B 0,C 180,E1 -19308.079,E2 -19308.079} C_VEL
LIN {X 0,Y 242.001,Z 351.341,A -85,B 0,C 180,E1 -19312.42,E2 -19312.42} C_VEL
LIN {X 0,Y 241.989,Z 351.34,A -85,B 0,C 180,E1 -19316.509,E2 -19316.509} C_VEL
LIN {X 0,Y 242.011,Z 351.341,A -85,B 0,C 180,E1 -19320.597,E2 -19320.597} C_VEL
LIN {X 0,Y 242.065,Z 351.329,A -85,B 0,C 180,E1 -19324.183,E2 -19324.183} C_VEL
LIN {X 0,Y 242.051,Z 351.334,A -85,B 0,C 180,E1 -19328.297,E2 -19328.297} C_VEL
LIN {X 0,Y 242.161,Z 351.316,A -85,B 0,C 180,E1 -19333.278,E2 -19333.278} C_VEL
LIN {X 0,Y 242.184,Z 351.318,A -85,B 0,C 180,E1 -19338.28,E2 -19338.28} C_VEL
LIN {X 0,Y 242.433,Z 351.282,A -85,B 0,C 180,E1 -19341.666,E2 -19341.666} C_VEL
LIN {X 0,Y 242.259,Z 351.307,A -85,B 0,C 180,E1 -19345.007,E2 -19345.007} C_VEL
LIN {X 0,Y 242.635,Z 351.262,A -85,B 0,C 180,E1 -19348.34,E2 -19348.34} C_VEL
LIN {X 0,Y 242.635,Z 351.258,A -85,B 0,C 180,E1 -19351.66,E2 -19351.66} C_VEL
LIN {X 0,Y 242.432,Z 351.285,A -85,B 0,C 180,E1 -19356.659,E2 -19356.659} C_VEL
LIN {X 0,Y 242.343,Z 351.296,A -85,B 0,C 180,E1 -19360.021,E2 -19360.021} C_VEL
LIN {X 0,Y 242.165,Z 351.317,A -85,B 0,C 180,E1 -19365.141,E2 -19365.141} C_VEL
LIN {X 0,Y 242.072,Z 351.33,A -85,B 0,C 180,E1 -19368.625,E2 -19368.625} C_VEL
LIN {X 0,Y 242.011,Z 351.341,A -85,B 0,C 180,E1 -19372.181,E2 -19372.181} C_VEL
LIN {X 0,Y 242.065,Z 351.329,A -85,B 0,C 180,E1 -19375.839,E2 -19375.839} C_VEL
LIN {X 0,Y 242.006,Z 351.338,A -85,B 0,C 180,E1 -19379.584,E2 -19379.584} C_VEL
LIN {X 0,Y 241.99,Z 351.338,A -85,B 0,C 180,E1 -19383.492,E2 -19383.492} C_VEL
LIN {X 0,Y 242.001,Z 351.339,A -85,B 0,C 180,E1 -19387.58,E2 -19387.58} C_VEL
LIN {X 0,Y 241.942,Z 351.347,A -85,B 0,C 180,E1 -19391.922,E2 -19391.922} C_VEL
LIN {X 0,Y 241.934,Z 351.347,A -85,B 0,C 180,E1 -19396.572,E2 -19396.572} C_VEL
LIN {X 0,Y 241.957,Z 351.343,A -85,B 0,C 180,E1 -19400.282,E2 -19400.282} C_VEL
LIN {X 0,Y 242.037,Z 351.335,A -85,B 0,C 180,E1 -19404.499,E2 -19404.499} C_VEL
LIN {X 0,Y 242.031,Z 351.335,A -85,B 0,C 180,E1 -19406.431,E2 -19406.431} C_VEL
LIN {X 0,Y 249.854,Z 376.369,A -85,B 0,C 180,E1 -19407.973,E2 -19407.973} C_VEL
LIN {X 0,Y 247.863,Z 433.878,A -85,B 0,C 180,E1 -19410.427,E2 -19410.427} C_VEL
LIN {X 0,Y 247.367,Z 447.908,A -85,B 0,C 180,E1 -19411.266,E2 -19411.266} C_VEL
LIN {X 0,Y 246.635,Z 461.725,A -85,B 0,C 180,E1 -19412.436,E2 -19412.436} C_VEL
LIN {X 0,Y 245.727,Z 474.908,A -85,B 0,C 180,E1 -19413.914,E2 -19413.914} C_VEL
LIN {X 0,Y 244.783,Z 486.82,A -85,B 0,C 180,E1 -19415.625,E2 -19415.625} C_VEL
LIN {X 0,Y 243.791,Z 498.373,A -85,B 0,C 180,E1 -19417.684,E2 -19417.684} C_VEL
LIN {X 0,Y 242.84,Z 509.295,A -85,B 0,C 180,E1 -19420.121,E2 -19420.121} C_VEL
LIN {X 0,Y 242.133,Z 518.511,A -85,B 0,C 180,E1 -19422.693,E2 -19422.693} C_VEL
LIN {X 0,Y 241.654,Z 525.884,A -85,B 0,C 180,E1 -19425.258,E2 -19425.258} C_VEL
LIN {X 0,Y 241.447,Z 530.864,A -85,B 0,C 180,E1 -19427.391,E2 -19427.391} C_VEL
LIN {X 0,Y 241.499,Z 535.697,A -85,B 0,C 180,E1 -19429.945,E2 -19429.945} C_VEL
LIN {X 0,Y 241.788,Z 539.364,A -85,B 0,C 180,E1 -19432.485,E2 -19432.485} C_VEL
LIN {X 0,Y 242.215,Z 541.987,A -85,B 0,C 180,E1 -19435.007,E2 -19435.007} C_VEL
LIN {X 0,Y 242.767,Z 543.157,A -85,B 0,C 180,E1 -19436.682,E2 -19436.682} C_VEL
LIN {X 0,Y 244.316,Z 544.275,A -85,B 0,C 180,E1 -19440.001,E2 -19440.001} C_VEL
LIN {X 0,Y 246.355,Z 543.714,A -85,B 0,C 180,E1 -19443.152,E2 -19443.152} C_VEL
LIN {X 0,Y 247.683,Z 542.755,A -85,B 0,C 180,E1 -19444.884,E2 -19444.884} C_VEL
LIN {X 0,Y 249.192,Z 541.404,A -85,B 0,C 180,E1 -19446.478,E2 -19446.478} C_VEL
LIN {X 0,Y 251.66,Z 538.564,A -85,B 0,C 180,E1 -19448.836,E2 -19448.836} C_VEL
LIN {X 0,Y 254.491,Z 534.632,A -85,B 0,C 180,E1 -19451.147,E2 -19451.147} C_VEL
LIN {X 0,Y 257.65,Z 529.54,A -85,B 0,C 180,E1 -19453.407,E2 -19453.407} C_VEL
LIN {X 0,Y 261.17,Z 523.188,A -85,B 0,C 180,E1 -19455.611,E2 -19455.611} C_VEL
LIN {X 0,Y 264.941,Z 515.31,A -85,B 0,C 180,E1 -19457.762,E2 -19457.762} C_VEL
LIN {X 0,Y 269.038,Z 505.495,A -85,B 0,C 180,E1 -19459.853,E2 -19459.853} C_VEL
LIN {X 0,Y 272.258,Z 496.597,A -85,B 0,C 180,E1 -19461.379,E2 -19461.379} C_VEL
LIN {X 0,Y 273.391,Z 492.169,A -85,B 0,C 180,E1 -19462.168,E2 -19462.168} C_VEL
LIN {X 0,Y 273.962,Z 485.124,A -85,B 0,C 180,E1 -19463.627,E2 -19463.627} C_VEL
LIN {X 0,Y 274.408,Z 477.711,A -85,B 0,C 180,E1 -19464.983,E2 -19464.983} C_VEL
LIN {X 0,Y 275.263,Z 472.72,A -85,B 0,C 180,E1 -19465.604,E2 -19465.604} C_VEL
LIN {X 0,Y 277.866,Z 459.877,A -85,B 0,C 180,E1 -19466.657,E2 -19466.657} C_VEL
LIN {X 0,Y 279.707,Z 447.141,A -85,B 0,C 180,E1 -19467.438,E2 -19467.438} C_VEL
LIN {X 0,Y 284.167,Z 416.621,A -85,B 0,C 180,E1 -19468.857,E2 -19468.857} C_VEL
LIN {X 0,Y 284.41,Z 415.01,A -85,B 0,C 180,E1 -19468.935,E2 -19468.935} C_VEL
LIN {X 0,Y 282.145,Z 410.116,A -85,B 0,C 180,E1 -19470.734,E2 -19470.734} C_VEL
LIN {X 0,Y 280.799,Z 407.454,A -85,B 0,C 180,E1 -19471.965,E2 -19471.965} C_VEL
LIN {X 0,Y 279.089,Z 404.038,A -85,B 0,C 180,E1 -19473.955,E2 -19473.955} C_VEL
LIN {X 0,Y 277.514,Z 401.158,A -85,B 0,C 180,E1 -19476.795,E2 -19476.795} C_VEL
LIN {X 0,Y 277.017,Z 400.695,A -85,B 0,C 180,E1 -19478.142,E2 -19478.142} C_VEL
LIN {X 0,Y 276.71,Z 401.101,A -85,B 0,C 180,E1 -19480.363,E2 -19480.363} C_VEL
LIN {X 0,Y 277.774,Z 403.631,A -85,B 0,C 180,E1 -19484.176,E2 -19484.176} C_VEL
LIN {X 0,Y 279.793,Z 408.143,A -85,B 0,C 180,E1 -19487.074,E2 -19487.074} C_VEL
LIN {X 0,Y 280.767,Z 410.471,A -85,B 0,C 180,E1 -19488.158,E2 -19488.158} C_VEL
LIN {X 0,Y 281.284,Z 415.597,A -85,B 0,C 180,E1 -19489.21,E2 -19489.21} C_VEL
LIN {X 0,Y 280.343,Z 431.411,A -85,B 0,C 180,E1 -19490.765,E2 -19490.765} C_VEL
LIN {X 0,Y 279.117,Z 450.407,A -85,B 0,C 180,E1 -19492.374,E2 -19492.374} C_VEL
LIN {X 0,Y 277.919,Z 464.803,A -85,B 0,C 180,E1 -19493.36,E2 -19493.36} C_VEL
LIN {X 0,Y 274.398,Z 487.064,A -85,B 0,C 180,E1 -19494.36,E2 -19494.36} C_VEL
LIN {X 0,Y 271.094,Z 501.634,A -85,B 0,C 180,E1 -19495.225,E2 -19495.225} C_VEL
LIN {X 0,Y 267.33,Z 514.747,A -85,B 0,C 180,E1 -19496.263,E2 -19496.263} C_VEL
LIN {X 0,Y 262.617,Z 528.109,A -85,B 0,C 180,E1 -19497.64,E2 -19497.64} C_VEL
LIN {X 0,Y 258.267,Z 539.151,A -85,B 0,C 180,E1 -19499.094,E2 -19499.094} C_VEL
LIN {X 0,Y 253.399,Z 550.19,A -85,B 0,C 180,E1 -19500.963,E2 -19500.963} C_VEL
LIN {X 0,Y 248.778,Z 560.181,A -85,B 0,C 180,E1 -19503.127,E2 -19503.127} C_VEL
LIN {X 0,Y 244.188,Z 569.629,A -85,B 0,C 180,E1 -19505.786,E2 -19505.786} C_VEL
LIN {X 0,Y 240.277,Z 577.309,A -85,B 0,C 180,E1 -19508.554,E2 -19508.554} C_VEL
LIN {X 0,Y 237.119,Z 583.834,A -85,B 0,C 180,E1 -19511.705,E2 -19511.705} C_VEL
LIN {X 0,Y 235.222,Z 588.044,A -85,B 0,C 180,E1 -19514.401,E2 -19514.401} C_VEL
LIN {X 0,Y 234.436,Z 590.168,A -85,B 0,C 180,E1 -19516.123,E2 -19516.123} C_VEL
LIN {X 0,Y 233.812,Z 591.868,A -85,B 0,C 180,E1 -19517.853,E2 -19517.853} C_VEL
LIN {X 0,Y 233.436,Z 594.07,A -85,B 0,C 180,E1 -19521.342,E2 -19521.342} C_VEL
LIN {X 0,Y 233.664,Z 594.607,A -85,B 0,C 180,E1 -19523.09,E2 -19523.09} C_VEL
LIN {X 0,Y 233.958,Z 594.735,A -85,B 0,C 180,E1 -19524.829,E2 -19524.829} C_VEL
LIN {X 0,Y 234.327,Z 594.404,A -85,B 0,C 180,E1 -19526.561,E2 -19526.561} C_VEL
LIN {X 0,Y 234.793,Z 593.624,A -85,B 0,C 180,E1 -19528.284,E2 -19528.284} C_VEL
LIN {X 0,Y 235.34,Z 592.449,A -85,B 0,C 180,E1 -19530.214,E2 -19530.214} C_VEL
LIN {X 0,Y 234.89,Z 593.673,A -85,B 0,C 180,E1 -19531.714,E2 -19531.714} C_VEL
LIN {X 0,Y 234.411,Z 594.638,A -85,B 0,C 180,E1 -19533.437,E2 -19533.437} C_VEL
LIN {X 0,Y 234.011,Z 595.143,A -85,B 0,C 180,E1 -19535.169,E2 -19535.169} C_VEL
LIN {X 0,Y 233.667,Z 595.222,A -85,B 0,C 180,E1 -19536.997,E2 -19536.997} C_VEL
LIN {X 0,Y 233.504,Z 594.227,A -85,B 0,C 180,E1 -19540.404,E2 -19540.404} C_VEL
LIN {X 0,Y 234.419,Z 591.723,A -85,B 0,C 180,E1 -19543.877,E2 -19543.877} C_VEL
LIN {X 0,Y 235.802,Z 588.835,A -85,B 0,C 180,E1 -19546.448,E2 -19546.448} C_VEL
LIN {X 0,Y 238.576,Z 583.578,A -85,B 0,C 180,E1 -19549.802,E2 -19549.802} C_VEL
LIN {X 0,Y 241.391,Z 578.528,A -85,B 0,C 180,E1 -19552.24,E2 -19552.24} C_VEL
LIN {X 0,Y 245.581,Z 571.267,A -85,B 0,C 180,E1 -19554.968,E2 -19554.968} C_VEL
LIN {X 0,Y 250.51,Z 562.374,A -85,B 0,C 180,E1 -19557.575,E2 -19557.575} C_VEL
LIN {X 0,Y 255.391,Z 553.105,A -85,B 0,C 180,E1 -19559.692,E2 -19559.692} C_VEL
LIN {X 0,Y 259.952,Z 543.976,A -85,B 0,C 180,E1 -19561.362,E2 -19561.362} C_VEL
LIN {X 0,Y 265.511,Z 532.051,A -85,B 0,C 180,E1 -19563.089,E2 -19563.089} C_VEL
LIN {X 0,Y 270.865,Z 518.858,A -85,B 0,C 180,E1 -19564.582,E2 -19564.582} C_VEL
LIN {X 0,Y 275.541,Z 505.854,A -85,B 0,C 180,E1 -19565.694,E2 -19565.694} C_VEL
LIN {X 0,Y 280.067,Z 490.488,A -85,B 0,C 180,E1 -19566.695,E2 -19566.695} C_VEL
LIN {X 0,Y 283.656,Z 474.009,A -85,B 0,C 180,E1 -19567.524,E2 -19567.524} C_VEL
LIN {X 0,Y 285.54,Z 462.785,A -85,B 0,C 180,E1 -19568.076,E2 -19568.076} C_VEL
LIN {X 0,Y 286.9,Z 451.163,A -85,B 0,C 180,E1 -19568.995,E2 -19568.995} C_VEL
LIN {X 0,Y 288.113,Z 437.814,A -85,B 0,C 180,E1 -19570.424,E2 -19570.424} C_VEL
LIN {X 0,Y 288.394,Z 433.726,A -85,B 0,C 180,E1 -19570.978,E2 -19570.978} C_VEL
LIN {X 0,Y 287.95,Z 430.705,A -85,B 0,C 180,E1 -19571.967,E2 -19571.967} C_VEL
LIN {X 0,Y 287.27,Z 425.088,A -85,B 0,C 180,E1 -19574.4,E2 -19574.4} C_VEL
LIN {X 0,Y 287.134,Z 422.096,A -85,B 0,C 180,E1 -19576.737,E2 -19576.737} C_VEL
LIN {X 0,Y 287.646,Z 420.551,A -85,B 0,C 180,E1 -19578.723,E2 -19578.723} C_VEL
LIN {X 0,Y 289.489,Z 420.796,A -85,B 0,C 180,E1 -19581.929,E2 -19581.929} C_VEL
LIN {X 0,Y 290.822,Z 422.01,A -85,B 0,C 180,E1 -19583.419,E2 -19583.419} C_VEL
LIN {X 0,Y 291.763,Z 423.23,A -85,B 0,C 180,E1 -19584.337,E2 -19584.337} C_VEL
LIN {X 0,Y 287.003,Z 448.986,A -85,B 0,C 180,E1 -19585.613,E2 -19585.613} C_VEL
LIN {X 0,Y 284.546,Z 462.458,A -85,B 0,C 180,E1 -19586.451,E2 -19586.451} C_VEL
LIN {X 0,Y 281.458,Z 475.345,A -85,B 0,C 180,E1 -19587.53,E2 -19587.53} C_VEL
LIN {X 0,Y 277.915,Z 487.109,A -85,B 0,C 180,E1 -19588.774,E2 -19588.774} C_VEL
LIN {X 0,Y 274.416,Z 496.752,A -85,B 0,C 180,E1 -19590.038,E2 -19590.038} C_VEL
LIN {X 0,Y 270.151,Z 506.831,A -85,B 0,C 180,E1 -19591.655,E2 -19591.655} C_VEL
LIN {X 0,Y 266.094,Z 515.2,A -85,B 0,C 180,E1 -19593.32,E2 -19593.32} C_VEL
LIN {X 0,Y 261.524,Z 523.444,A -85,B 0,C 180,E1 -19595.383,E2 -19595.383} C_VEL
LIN {X 0,Y 257.227,Z 530.21,A -85,B 0,C 180,E1 -19597.51,E2 -19597.51} C_VEL
LIN {X 0,Y 253.306,Z 535.642,A -85,B 0,C 180,E1 -19599.707,E2 -19599.707} C_VEL
LIN {X 0,Y 249.705,Z 539.922,A -85,B 0,C 180,E1 -19601.964,E2 -19601.964} C_VEL
LIN {X 0,Y 247.5,Z 542.172,A -85,B 0,C 180,E1 -19603.503,E2 -19603.503} C_VEL
LIN {X 0,Y 243.582,Z 545.391,A -85,B 0,C 180,E1 -19606.654,E2 -19606.654} C_VEL
LIN {X 0,Y 241.918,Z 546.356,A -85,B 0,C 180,E1 -19608.266,E2 -19608.266} C_VEL
LIN {X 0,Y 240.382,Z 546.905,A -85,B 0,C 180,E1 -19609.896,E2 -19609.896} C_VEL
LIN {X 0,Y 237.942,Z 546.806,A -85,B 0,C 180,E1 -19613.214,E2 -19613.214} C_VEL
LIN {X 0,Y 236.913,Z 546.147,A -85,B 0,C 180,E1 -19614.893,E2 -19614.893} C_VEL
LIN {X 0,Y 235.461,Z 543.561,A -85,B 0,C 180,E1 -19618.289,E2 -19618.289} C_VEL
LIN {X 0,Y 234.664,Z 540.521,A -85,B 0,C 180,E1 -19620.857,E2 -19620.857} C_VEL
LIN {X 0,Y 234.223,Z 536.445,A -85,B 0,C 180,E1 -19623.44,E2 -19623.44} C_VEL
LIN {X 0,Y 234.423,Z 530.29,A -85,B 0,C 180,E1 -19626.454,E2 -19626.454} C_VEL
LIN {X 0,Y 234.672,Z 522.289,A -85,B 0,C 180,E1 -19629.48,E2 -19629.48} C_VEL
LIN {X 0,Y 235.16,Z 513.735,A -85,B 0,C 180,E1 -19632.075,E2 -19632.075} C_VEL
LIN {X 0,Y 235.903,Z 503.118,A -85,B 0,C 180,E1 -19634.668,E2 -19634.668} C_VEL
LIN {X 0,Y 236.654,Z 493.408,A -85,B 0,C 180,E1 -19636.608,E2 -19636.608} C_VEL
LIN {X 0,Y 237.554,Z 481.234,A -85,B 0,C 180,E1 -19638.59,E2 -19638.59} C_VEL
LIN {X 0,Y 238.47,Z 468.372,A -85,B 0,C 180,E1 -19640.259,E2 -19640.259} C_VEL
LIN {X 0,Y 239.216,Z 454.377,A -85,B 0,C 180,E1 -19641.658,E2 -19641.658} C_VEL
LIN {X 0,Y 239.874,Z 440.366,A -85,B 0,C 180,E1 -19642.672,E2 -19642.672} C_VEL
LIN {X 0,Y 241.664,Z 385.519,A -85,B 0,C 180,E1 -19645.324,E2 -19645.324} C_VEL
LIN {X 0,Y 241.926,Z 376.15,A -85,B 0,C 180,E1 -19645.769,E2 -19645.769} C_VEL
LIN {X 0,Y 235.042,Z 352.206,A -85,B 0,C 180,E1 -19647.252,E2 -19647.252} C_VEL
LIN {X 0,Y 234.931,Z 352.218,A -85,B 0,C 180,E1 -19650.567,E2 -19650.567} C_VEL
LIN {X 0,Y 234.929,Z 352.222,A -85,B 0,C 180,E1 -19654.637,E2 -19654.637} C_VEL
LIN {X 0,Y 234.94,Z 352.219,A -85,B 0,C 180,E1 -19658.944,E2 -19658.944} C_VEL
LIN {X 0,Y 234.888,Z 352.224,A -85,B 0,C 180,E1 -19663.485,E2 -19663.485} C_VEL
LIN {X 0,Y 234.888,Z 352.225,A -85,B 0,C 180,E1 -19666.514,E2 -19666.514} C_VEL
LIN {X 0,Y 234.953,Z 352.218,A -85,B 0,C 180,E1 -19671.086,E2 -19671.086} C_VEL
LIN {X 0,Y 234.958,Z 352.213,A -85,B 0,C 180,E1 -19675.367,E2 -19675.367} C_VEL
LIN {X 0,Y 234.92,Z 352.22,A -85,B 0,C 180,E1 -19679.431,E2 -19679.431} C_VEL
LIN {X 0,Y 234.991,Z 352.209,A -85,B 0,C 180,E1 -19683.794,E2 -19683.794} C_VEL
LIN {X 0,Y 235.009,Z 352.21,A -85,B 0,C 180,E1 -19688.97,E2 -19688.97} C_VEL
LIN {X 0,Y 235.094,Z 352.197,A -85,B 0,C 180,E1 -19693.059,E2 -19693.059} C_VEL
LIN {X 0,Y 235.144,Z 352.193,A -85,B 0,C 180,E1 -19697.924,E2 -19697.924} C_VEL
LIN {X 0,Y 235.388,Z 352.159,A -85,B 0,C 180,E1 -19701.415,E2 -19701.415} C_VEL
LIN {X 0,Y 235.403,Z 352.16,A -85,B 0,C 180,E1 -19703.142,E2 -19703.142} C_VEL
LIN {X 0,Y 235.594,Z 352.139,A -85,B 0,C 180,E1 -19708.291,E2 -19708.291} C_VEL
LIN {X 0,Y 235.594,Z 352.135,A -85,B 0,C 180,E1 -19711.71,E2 -19711.71} C_VEL
LIN {X 0,Y 235.404,Z 352.159,A -85,B 0,C 180,E1 -19716.859,E2 -19716.859} C_VEL
LIN {X 0,Y 235.251,Z 352.181,A -85,B 0,C 180,E1 -19720.326,E2 -19720.326} C_VEL
LIN {X 0,Y 235.112,Z 352.196,A -85,B 0,C 180,E1 -19725.607,E2 -19725.607} C_VEL
LIN {X 0,Y 235.007,Z 352.209,A -85,B 0,C 180,E1 -19729.206,E2 -19729.206} C_VEL
LIN {X 0,Y 234.959,Z 352.215,A -85,B 0,C 180,E1 -19732.883,E2 -19732.883} C_VEL
LIN {X 0,Y 234.966,Z 352.214,A -85,B 0,C 180,E1 -19736.658,E2 -19736.658} C_VEL
LIN {X 0,Y 234.921,Z 352.221,A -85,B 0,C 180,E1 -19740.57,E2 -19740.57} C_VEL
LIN {X 0,Y 234.96,Z 352.214,A -85,B 0,C 180,E1 -19744.634,E2 -19744.634} C_VEL
LIN {X 0,Y 234.941,Z 352.218,A -85,B 0,C 180,E1 -19748.945,E2 -19748.945} C_VEL
LIN {X 0,Y 234.886,Z 352.223,A -85,B 0,C 180,E1 -19753.487,E2 -19753.487} C_VEL
LIN {X 0,Y 234.887,Z 352.226,A -85,B 0,C 180,E1 -19756.515,E2 -19756.515} C_VEL
LIN {X 0,Y 234.92,Z 352.217,A -85,B 0,C 180,E1 -19761.08,E2 -19761.08} C_VEL
LIN {X 0,Y 235.009,Z 352.21,A -85,B 0,C 180,E1 -19765.376,E2 -19765.376} C_VEL
LIN {X 0,Y 235.02,Z 352.297,A -85,B 0,C 180,E1 -19766.129,E2 -19766.129} C_VEL
LIN {X 0,Y 242.821,Z 377.494,A -85,B 0,C 180,E1 -19767.7,E2 -19767.7} C_VEL
LIN {X 0,Y 240.858,Z 433.973,A -85,B 0,C 180,E1 -19770.202,E2 -19770.202} C_VEL
LIN {X 0,Y 240.328,Z 448.081,A -85,B 0,C 180,E1 -19771.053,E2 -19771.053} C_VEL
LIN {X 0,Y 239.579,Z 462.002,A -85,B 0,C 180,E1 -19772.246,E2 -19772.246} C_VEL
LIN {X 0,Y 238.634,Z 475.433,A -85,B 0,C 180,E1 -19773.784,E2 -19773.784} C_VEL
LIN {X 0,Y 237.71,Z 487.463,A -85,B 0,C 180,E1 -19775.55,E2 -19775.55} C_VEL
LIN {X 0,Y 236.741,Z 498.353,A -85,B 0,C 180,E1 -19777.53,E2 -19777.53} C_VEL
LIN {X 0,Y 235.937,Z 507.304,A -85,B 0,C 180,E1 -19779.513,E2 -19779.513} C_VEL
LIN {X 0,Y 235.161,Z 517.068,A -85,B 0,C 180,E1 -19782.163,E2 -19782.163} C_VEL
LIN {X 0,Y 234.644,Z 524.919,A -85,B 0,C 180,E1 -19784.807,E2 -19784.807} C_VEL
LIN {X 0,Y 234.346,Z 532.134,A -85,B 0,C 180,E1 -19787.883,E2 -19787.883} C_VEL
LIN {X 0,Y 234.468,Z 536.92,A -85,B 0,C 180,E1 -19790.513,E2 -19790.513} C_VEL
LIN {X 0,Y 234.782,Z 540.529,A -85,B 0,C 180,E1 -19793.124,E2 -19793.124} C_VEL
LIN {X 0,Y 235.09,Z 542.336,A -85,B 0,C 180,E1 -19794.855,E2 -19794.855} C_VEL
LIN {X 0,Y 235.639,Z 543.734,A -85,B 0,C 180,E1 -19796.581,E2 -19796.581} C_VEL
LIN {X 0,Y 236.351,Z 544.717,A -85,B 0,C 180,E1 -19798.297,E2 -19798.297} C_VEL
LIN {X 0,Y 237.234,Z 545.231,A -85,B 0,C 180,E1 -19800.001,E2 -19800.001} C_VEL
LIN {X 0,Y 239.456,Z 545.062,A -85,B 0,C 180,E1 -19803.366,E2 -19803.366} C_VEL
LIN {X 0,Y 240.728,Z 544.353,A -85,B 0,C 180,E1 -19805.025,E2 -19805.025} C_VEL
LIN {X 0,Y 242.294,Z 543.192,A -85,B 0,C 180,E1 -19806.663,E2 -19806.663} C_VEL
LIN {X 0,Y 244.864,Z 540.664,A -85,B 0,C 180,E1 -19809.083,E2 -19809.083} C_VEL
LIN {X 0,Y 247.819,Z 537.116,A -85,B 0,C 180,E1 -19811.451,E2 -19811.451} C_VEL
LIN {X 0,Y 251.121,Z 532.472,A -85,B 0,C 180,E1 -19813.763,E2 -19813.763} C_VEL
LIN {X 0,Y 254.742,Z 526.579,A -85,B 0,C 180,E1 -19816.016,E2 -19816.016} C_VEL
LIN {X 0,Y 258.707,Z 519.249,A -85,B 0,C 180,E1 -19818.206,E2 -19818.206} C_VEL
LIN {X 0,Y 263.018,Z 510.172,A -85,B 0,C 180,E1 -19820.327,E2 -19820.327} C_VEL
LIN {X 0,Y 267.121,Z 499.907,A -85,B 0,C 180,E1 -19822.224,E2 -19822.224} C_VEL
LIN {X 0,Y 270.883,Z 489.018,A -85,B 0,C 180,E1 -19823.815,E2 -19823.815} C_VEL
LIN {X 0,Y 274.306,Z 476.722,A -85,B 0,C 180,E1 -19825.211,E2 -19825.211} C_VEL
LIN {X 0,Y 275.263,Z 472.72,A -85,B 0,C 180,E1 -19825.604,E2 -19825.604} C_VEL
LIN {X 0,Y 276.084,Z 467.596,A -85,B 0,C 180,E1 -19826.196,E2 -19826.196} C_VEL
LIN {X 0,Y 276.284,Z 459.466,A -85,B 0,C 180,E1 -19827.379,E2 -19827.379} C_VEL
LIN {X 0,Y 276.354,Z 451.097,A -85,B 0,C 180,E1 -19828.451,E2 -19828.451} C_VEL
LIN {X 0,Y 276.872,Z 445.622,A -85,B 0,C 180,E1 -19828.865,E2 -19828.865} C_VEL
LIN {X 0,Y 281.012,Z 419.21,A -85,B 0,C 180,E1 -19830.094,E2 -19830.094} C_VEL
LIN {X 0,Y 278.79,Z 414.16,A -85,B 0,C 180,E1 -19832.223,E2 -19832.223} C_VEL
LIN {X 0,Y 277.076,Z 410.577,A -85,B 0,C 180,E1 -19834.39,E2 -19834.39} C_VEL
LIN {X 0,Y 275.754,Z 407.934,A -85,B 0,C 180,E1 -19837.069,E2 -19837.069} C_VEL
LIN {X 0,Y 275.499,Z 407.674,A -85,B 0,C 180,E1 -19837.753,E2 -19837.753} C_VEL
LIN {X 0,Y 275.059,Z 407.949,A -85,B 0,C 180,E1 -19840.175,E2 -19840.175} C_VEL
LIN {X 0,Y 275.955,Z 410.427,A -85,B 0,C 180,E1 -19843.922,E2 -19843.922} C_VEL
LIN {X 0,Y 277.798,Z 414.851,A -85,B 0,C 180,E1 -19846.79,E2 -19846.79} C_VEL
LIN {X 0,Y 278.306,Z 416.424,A -85,B 0,C 180,E1 -19847.462,E2 -19847.462} C_VEL
LIN {X 0,Y 278.474,Z 419.646,A -85,B 0,C 180,E1 -19848.13,E2 -19848.13} C_VEL
LIN {X 0,Y 277.103,Z 436.811,A -85,B 0,C 180,E1 -19849.818,E2 -19849.818} C_VEL
LIN {X 0,Y 275.55,Z 455.794,A -85,B 0,C 180,E1 -19851.411,E2 -19851.411} C_VEL
LIN {X 0,Y 274.485,Z 465.813,A -85,B 0,C 180,E1 -19852.084,E2 -19852.084} C_VEL
LIN {X 0,Y 270.978,Z 486.608,A -85,B 0,C 180,E1 -19853.03,E2 -19853.03} C_VEL
LIN {X 0,Y 267.239,Z 501.713,A -85,B 0,C 180,E1 -19853.954,E2 -19853.954} C_VEL
LIN {X 0,Y 263.289,Z 514.332,A -85,B 0,C 180,E1 -19854.977,E2 -19854.977} C_VEL
LIN {X 0,Y 258.368,Z 527.581,A -85,B 0,C 180,E1 -19856.342,E2 -19856.342} C_VEL
LIN {X 0,Y 253.292,Z 539.409,A -85,B 0,C 180,E1 -19857.95,E2 -19857.95} C_VEL
LIN {X 0,Y 248.183,Z 550.193,A -85,B 0,C 180,E1 -19859.825,E2 -19859.825} C_VEL
LIN {X 0,Y 243.268,Z 559.873,A -85,B 0,C 180,E1 -19862,E2 -19862} C_VEL
LIN {X 0,Y 238.407,Z 569.133,A -85,B 0,C 180,E1 -19864.694,E2 -19864.694} C_VEL
LIN {X 0,Y 234.755,Z 575.655,A -85,B 0,C 180,E1 -19867.095,E2 -19867.095} C_VEL
LIN {X 0,Y 231.787,Z 580.997,A -85,B 0,C 180,E1 -19869.592,E2 -19869.592} C_VEL
LIN {X 0,Y 229.593,Z 585.328,A -85,B 0,C 180,E1 -19872.175,E2 -19872.175} C_VEL
LIN {X 0,Y 228.349,Z 587.682,A -85,B 0,C 180,E1 -19873.919,E2 -19873.919} C_VEL
LIN {X 0,Y 226.822,Z 591.177,A -85,B 0,C 180,E1 -19877.473,E2 -19877.473} C_VEL
LIN {X 0,Y 226.386,Z 593.173,A -85,B 0,C 180,E1 -19881.07,E2 -19881.07} C_VEL
LIN {X 0,Y 226.6,Z 593.577,A -85,B 0,C 180,E1 -19882.974,E2 -19882.974} C_VEL
LIN {X 0,Y 226.916,Z 593.551,A -85,B 0,C 180,E1 -19884.668,E2 -19884.668} C_VEL
LIN {X 0,Y 227.31,Z 593.116,A -85,B 0,C 180,E1 -19886.454,E2 -19886.454} C_VEL
LIN {X 0,Y 227.8,Z 592.268,A -85,B 0,C 180,E1 -19888.232,E2 -19888.232} C_VEL
LIN {X 0,Y 228.435,Z 590.788,A -85,B 0,C 180,E1 -19890.22,E2 -19890.22} C_VEL
LIN {X 0,Y 227.957,Z 592.113,A -85,B 0,C 180,E1 -19891.766,E2 -19891.766} C_VEL
LIN {X 0,Y 227.434,Z 593.181,A -85,B 0,C 180,E1 -19893.543,E2 -19893.543} C_VEL
LIN {X 0,Y 226.983,Z 593.825,A -85,B 0,C 180,E1 -19895.329,E2 -19895.329} C_VEL
LIN {X 0,Y 226.649,Z 594.056,A -85,B 0,C 180,E1 -19897.125,E2 -19897.125} C_VEL
LIN {X 0,Y 226.501,Z 593.299,A -85,B 0,C 180,E1 -19900.729,E2 -19900.729} C_VEL
LIN {X 0,Y 227.498,Z 591.073,A -85,B 0,C 180,E1 -19904.308,E2 -19904.308} C_VEL
LIN {X 0,Y 229.617,Z 587.381,A -85,B 0,C 180,E1 -19907.823,E2 -19907.823} C_VEL
LIN {X 0,Y 231.883,Z 583.56,A -85,B 0,C 180,E1 -19910.398,E2 -19910.398} C_VEL
LIN {X 0,Y 234.861,Z 578.822,A -85,B 0,C 180,E1 -19912.893,E2 -19912.893} C_VEL
LIN {X 0,Y 239.225,Z 572.022,A -85,B 0,C 180,E1 -19915.679,E2 -19915.679} C_VEL
LIN {X 0,Y 244.339,Z 563.627,A -85,B 0,C 180,E1 -19918.333,E2 -19918.333} C_VEL
LIN {X 0,Y 249.368,Z 554.954,A -85,B 0,C 180,E1 -19920.484,E2 -19920.484} C_VEL
LIN {X 0,Y 255.054,Z 544.609,A -85,B 0,C 180,E1 -19922.501,E2 -19922.501} C_VEL
LIN {X 0,Y 260.837,Z 533.131,A -85,B 0,C 180,E1 -19924.226,E2 -19924.226} C_VEL
LIN {X 0,Y 266.418,Z 520.669,A -85,B 0,C 180,E1 -19925.708,E2 -19925.708} C_VEL
LIN {X 0,Y 271.22,Z 508.49,A -85,B 0,C 180,E1 -19926.815,E2 -19926.815} C_VEL
LIN {X 0,Y 276.228,Z 493.413,A -85,B 0,C 180,E1 -19927.865,E2 -19927.865} C_VEL
LIN {X 0,Y 280.417,Z 476.929,A -85,B 0,C 180,E1 -19928.74,E2 -19928.74} C_VEL
LIN {X 0,Y 282.912,Z 463.563,A -85,B 0,C 180,E1 -19929.401,E2 -19929.401} C_VEL
LIN {X 0,Y 284.287,Z 453.209,A -85,B 0,C 180,E1 -19930.263,E2 -19930.263} C_VEL
LIN {X 0,Y 285.714,Z 440.852,A -85,B 0,C 180,E1 -19931.617,E2 -19931.617} C_VEL
LIN {X 0,Y 285.909,Z 438.348,A -85,B 0,C 180,E1 -19932.006,E2 -19932.006} C_VEL
LIN {X 0,Y 285.462,Z 434.322,A -85,B 0,C 180,E1 -19933.579,E2 -19933.579} C_VEL
LIN {X 0,Y 285.336,Z 431.512,A -85,B 0,C 180,E1 -19934.863,E2 -19934.863} C_VEL
LIN {X 0,Y 285.38,Z 428.734,A -85,B 0,C 180,E1 -19937.094,E2 -19937.094} C_VEL
LIN {X 0,Y 285.954,Z 427.361,A -85,B 0,C 180,E1 -19938.983,E2 -19938.983} C_VEL
LIN {X 0,Y 288.026,Z 427.821,A -85,B 0,C 180,E1 -19942.302,E2 -19942.302} C_VEL
LIN {X 0,Y 288.77,Z 428.884,A -85,B 0,C 180,E1 -19943.223,E2 -19943.223} C_VEL
LIN {X 0,Y 283.704,Z 455.006,A -85,B 0,C 180,E1 -19944.568,E2 -19944.568} C_VEL
LIN {X 0,Y 281.279,Z 466.509,A -85,B 0,C 180,E1 -19945.359,E2 -19945.359} C_VEL
LIN {X 0,Y 277.962,Z 478.798,A -85,B 0,C 180,E1 -19946.42,E2 -19946.42} C_VEL
LIN {X 0,Y 273.261,Z 492.504,A -85,B 0,C 180,E1 -19947.963,E2 -19947.963} C_VEL
LIN {X 0,Y 268.245,Z 504.405,A -85,B 0,C 180,E1 -19949.711,E2 -19949.711} C_VEL
LIN {X 0,Y 262.972,Z 514.896,A -85,B 0,C 180,E1 -19951.681,E2 -19951.681} C_VEL
LIN {X 0,Y 258.017,Z 523.435,A -85,B 0,C 180,E1 -19953.728,E2 -19953.728} C_VEL
LIN {X 0,Y 252.618,Z 531.381,A -85,B 0,C 180,E1 -19956.208,E2 -19956.208} C_VEL
LIN {X 0,Y 248.412,Z 536.777,A -85,B 0,C 180,E1 -19958.42,E2 -19958.42} C_VEL
LIN {X 0,Y 244.508,Z 541.05,A -85,B 0,C 180,E1 -19960.697,E2 -19960.697} C_VEL
LIN {X 0,Y 241,Z 544.273,A -85,B 0,C 180,E1 -19963.044,E2 -19963.044} C_VEL
LIN {X 0,Y 238.856,Z 545.893,A -85,B 0,C 180,E1 -19964.643,E2 -19964.643} C_VEL
LIN {X 0,Y 236.866,Z 547.068,A -85,B 0,C 180,E1 -19966.268,E2 -19966.268} C_VEL
LIN {X 0,Y 233.523,Z 548.227,A -85,B 0,C 180,E1 -19969.596,E2 -19969.596} C_VEL
LIN {X 0,Y 232.187,Z 548.184,A -85,B 0,C 180,E1 -19971.294,E2 -19971.294} C_VEL
LIN {X 0,Y 229.881,Z 546.892,A -85,B 0,C 180,E1 -19974.737,E2 -19974.737} C_VEL
LIN {X 0,Y 229.072,Z 545.651,A -85,B 0,C 180,E1 -19976.481,E2 -19976.481} C_VEL
LIN {X 0,Y 228.084,Z 542.984,A -85,B 0,C 180,E1 -19979.116,E2 -19979.116} C_VEL
LIN {X 0,Y 227.342,Z 539.328,A -85,B 0,C 180,E1 -19981.771,E2 -19981.771} C_VEL
LIN {X 0,Y 227.156,Z 534.607,A -85,B 0,C 180,E1 -19984.435,E2 -19984.435} C_VEL
LIN {X 0,Y 227.334,Z 528.313,A -85,B 0,C 180,E1 -19987.25,E2 -19987.25} C_VEL
LIN {X 0,Y 227.741,Z 519.988,A -85,B 0,C 180,E1 -19990.22,E2 -19990.22} C_VEL
LIN {X 0,Y 228.15,Z 512.344,A -85,B 0,C 180,E1 -19992.452,E2 -19992.452} C_VEL
LIN {X 0,Y 228.884,Z 502.191,A -85,B 0,C 180,E1 -19994.901,E2 -19994.901} C_VEL
LIN {X 0,Y 229.796,Z 490.905,A -85,B 0,C 180,E1 -19997.119,E2 -19997.119} C_VEL
LIN {X 0,Y 230.619,Z 479.453,A -85,B 0,C 180,E1 -19998.942,E2 -19998.942} C_VEL
LIN {X 0,Y 231.54,Z 465.866,A -85,B 0,C 180,E1 -20000.661,E2 -20000.661} C_VEL
LIN {X 0,Y 232.299,Z 452.048,A -85,B 0,C 180,E1 -20001.986,E2 -20001.986} C_VEL
LIN {X 0,Y 232.893,Z 438.85,A -85,B 0,C 180,E1 -20002.921,E2 -20002.921} C_VEL
LIN {X 0,Y 234.643,Z 385.581,A -85,B 0,C 180,E1 -20005.574,E2 -20005.574} C_VEL
LIN {X 0,Y 234.99,Z 377.626,A -85,B 0,C 180,E1 -20005.961,E2 -20005.961} C_VEL
LIN {X 0,Y 227.98,Z 353.084,A -85,B 0,C 180,E1 -20007.542,E2 -20007.542} C_VEL
LIN {X 0,Y 227.87,Z 353.098,A -85,B 0,C 180,E1 -20011.621,E2 -20011.621} C_VEL
LIN {X 0,Y 227.879,Z 353.097,A -85,B 0,C 180,E1 -20015.871,E2 -20015.871} C_VEL
LIN {X 0,Y 227.825,Z 353.104,A -85,B 0,C 180,E1 -20020.376,E2 -20020.376} C_VEL
LIN {X 0,Y 227.833,Z 353.103,A -85,B 0,C 180,E1 -20025.192,E2 -20025.192} C_VEL
LIN {X 0,Y 227.832,Z 353.103,A -85,B 0,C 180,E1 -20029.625,E2 -20029.625} C_VEL
LIN {X 0,Y 227.898,Z 353.095,A -85,B 0,C 180,E1 -20034.131,E2 -20034.131} C_VEL
LIN {X 0,Y 227.867,Z 353.1,A -85,B 0,C 180,E1 -20038.377,E2 -20038.377} C_VEL
LIN {X 0,Y 227.877,Z 353.1,A -85,B 0,C 180,E1 -20042.444,E2 -20042.444} C_VEL
LIN {X 0,Y 227.912,Z 353.094,A -85,B 0,C 180,E1 -20046.367,E2 -20046.367} C_VEL
LIN {X 0,Y 227.94,Z 353.091,A -85,B 0,C 180,E1 -20050.175,E2 -20050.175} C_VEL
LIN {X 0,Y 228.055,Z 353.074,A -85,B 0,C 180,E1 -20053.898,E2 -20053.898} C_VEL
LIN {X 0,Y 228.169,Z 353.06,A -85,B 0,C 180,E1 -20059.35,E2 -20059.35} C_VEL
LIN {X 0,Y 228.356,Z 353.038,A -85,B 0,C 180,E1 -20062.929,E2 -20062.929} C_VEL
LIN {X 0,Y 228.553,Z 353.016,A -85,B 0,C 180,E1 -20068.238,E2 -20068.238} C_VEL
LIN {X 0,Y 228.553,Z 353.013,A -85,B 0,C 180,E1 -20071.762,E2 -20071.762} C_VEL
LIN {X 0,Y 228.356,Z 353.036,A -85,B 0,C 180,E1 -20077.072,E2 -20077.072} C_VEL
LIN {X 0,Y 228.17,Z 353.063,A -85,B 0,C 180,E1 -20080.65,E2 -20080.65} C_VEL
LIN {X 0,Y 228.056,Z 353.077,A -85,B 0,C 180,E1 -20086.103,E2 -20086.103} C_VEL
LIN {X 0,Y 227.941,Z 353.09,A -85,B 0,C 180,E1 -20089.826,E2 -20089.826} C_VEL
LIN {X 0,Y 227.912,Z 353.093,A -85,B 0,C 180,E1 -20093.633,E2 -20093.633} C_VEL
LIN {X 0,Y 227.878,Z 353.097,A -85,B 0,C 180,E1 -20097.557,E2 -20097.557} C_VEL
LIN {X 0,Y 227.868,Z 353.099,A -85,B 0,C 180,E1 -20101.623,E2 -20101.623} C_VEL
LIN {X 0,Y 227.899,Z 353.095,A -85,B 0,C 180,E1 -20105.869,E2 -20105.869} C_VEL
LIN {X 0,Y 227.832,Z 353.104,A -85,B 0,C 180,E1 -20110.376,E2 -20110.376} C_VEL
LIN {X 0,Y 227.833,Z 353.103,A -85,B 0,C 180,E1 -20115.194,E2 -20115.194} C_VEL
LIN {X 0,Y 227.826,Z 353.105,A -85,B 0,C 180,E1 -20119.624,E2 -20119.624} C_VEL
LIN {X 0,Y 227.908,Z 353.097,A -85,B 0,C 180,E1 -20124.134,E2 -20124.134} C_VEL
LIN {X 0,Y 227.973,Z 353.088,A -85,B 0,C 180,E1 -20125.741,E2 -20125.741} C_VEL
LIN {X 0,Y 235.871,Z 379.542,A -85,B 0,C 180,E1 -20127.469,E2 -20127.469} C_VEL
LIN {X 0,Y 233.833,Z 433.399,A -85,B 0,C 180,E1 -20129.93,E2 -20129.93} C_VEL
LIN {X 0,Y 233.359,Z 447.451,A -85,B 0,C 180,E1 -20130.772,E2 -20130.772} C_VEL
LIN {X 0,Y 232.59,Z 461.149,A -85,B 0,C 180,E1 -20131.951,E2 -20131.951} C_VEL
LIN {X 0,Y 231.717,Z 474.037,A -85,B 0,C 180,E1 -20133.426,E2 -20133.426} C_VEL
LIN {X 0,Y 230.704,Z 486.498,A -85,B 0,C 180,E1 -20135.238,E2 -20135.238} C_VEL
LIN {X 0,Y 229.621,Z 498.792,A -85,B 0,C 180,E1 -20137.507,E2 -20137.507} C_VEL
LIN {X 0,Y 228.727,Z 508.741,A -85,B 0,C 180,E1 -20139.778,E2 -20139.778} C_VEL
LIN {X 0,Y 228.091,Z 516.96,A -85,B 0,C 180,E1 -20142.055,E2 -20142.055} C_VEL
LIN {X 0,Y 227.543,Z 525.06,A -85,B 0,C 180,E1 -20144.78,E2 -20144.78} C_VEL
LIN {X 0,Y 227.265,Z 531.51,A -85,B 0,C 180,E1 -20147.499,E2 -20147.499} C_VEL
LIN {X 0,Y 227.343,Z 536.613,A -85,B 0,C 180,E1 -20150.212,E2 -20150.212} C_VEL
LIN {X 0,Y 227.673,Z 540.557,A -85,B 0,C 180,E1 -20152.908,E2 -20152.908} C_VEL
LIN {X 0,Y 227.972,Z 542.62,A -85,B 0,C 180,E1 -20154.694,E2 -20154.694} C_VEL
LIN {X 0,Y 228.504,Z 544.226,A -85,B 0,C 180,E1 -20156.474,E2 -20156.474} C_VEL
LIN {X 0,Y 229.249,Z 545.375,A -85,B 0,C 180,E1 -20158.244,E2 -20158.244} C_VEL
LIN {X 0,Y 230.156,Z 546.121,A -85,B 0,C 180,E1 -20160.001,E2 -20160.001} C_VEL
LIN {X 0,Y 231.186,Z 546.467,A -85,B 0,C 180,E1 -20161.743,E2 -20161.743} C_VEL
LIN {X 0,Y 232.441,Z 546.346,A -85,B 0,C 180,E1 -20163.468,E2 -20163.468} C_VEL
LIN {X 0,Y 233.759,Z 545.849,A -85,B 0,C 180,E1 -20165.176,E2 -20165.176} C_VEL
LIN {X 0,Y 235.388,Z 544.924,A -85,B 0,C 180,E1 -20166.86,E2 -20166.86} C_VEL
LIN {X 0,Y 237.148,Z 543.566,A -85,B 0,C 180,E1 -20168.522,E2 -20168.522} C_VEL
LIN {X 0,Y 240.062,Z 540.747,A -85,B 0,C 180,E1 -20170.971,E2 -20170.971} C_VEL
LIN {X 0,Y 243.368,Z 536.846,A -85,B 0,C 180,E1 -20173.358,E2 -20173.358} C_VEL
LIN {X 0,Y 247.08,Z 531.789,A -85,B 0,C 180,E1 -20175.678,E2 -20175.678} C_VEL
LIN {X 0,Y 251.339,Z 525.104,A -85,B 0,C 180,E1 -20178.061,E2 -20178.061} C_VEL
LIN {X 0,Y 255.461,Z 517.666,A -85,B 0,C 180,E1 -20180.115,E2 -20180.115} C_VEL
LIN {X 0,Y 260.075,Z 508.069,A -85,B 0,C 180,E1 -20182.231,E2 -20182.231} C_VEL
LIN {X 0,Y 264.163,Z 498.111,A -85,B 0,C 180,E1 -20183.937,E2 -20183.937} C_VEL
LIN {X 0,Y 267.995,Z 487.248,A -85,B 0,C 180,E1 -20185.432,E2 -20185.432} C_VEL
LIN {X 0,Y 271.393,Z 475.263,A -85,B 0,C 180,E1 -20186.741,E2 -20186.741} C_VEL
LIN {X 0,Y 274.254,Z 462.298,A -85,B 0,C 180,E1 -20187.838,E2 -20187.838} C_VEL
LIN {X 0,Y 276.27,Z 449.981,A -85,B 0,C 180,E1 -20188.629,E2 -20188.629} C_VEL
LIN {X 0,Y 276.872,Z 445.622,A -85,B 0,C 180,E1 -20188.865,E2 -20188.865} C_VEL
LIN {X 0,Y 277.159,Z 441.931,A -85,B 0,C 180,E1 -20189.182,E2 -20189.182} C_VEL
LIN {X 0,Y 276.81,Z 431.018,A -85,B 0,C 180,E1 -20190.839,E2 -20190.839} C_VEL
LIN {X 0,Y 277.257,Z 427.316,A -85,B 0,C 180,E1 -20191.115,E2 -20191.115} C_VEL
LIN {X 0,Y 277.861,Z 423.529,A -85,B 0,C 180,E1 -20191.323,E2 -20191.323} C_VEL
LIN {X 0,Y 276.3,Z 419.946,A -85,B 0,C 180,E1 -20193.062,E2 -20193.062} C_VEL
LIN {X 0,Y 275.215,Z 417.312,A -85,B 0,C 180,E1 -20194.655,E2 -20194.655} C_VEL
LIN {X 0,Y 274.003,Z 414.724,A -85,B 0,C 180,E1 -20197.331,E2 -20197.331} C_VEL
LIN {X 0,Y 273.409,Z 414.78,A -85,B 0,C 180,E1 -20199.989,E2 -20199.989} C_VEL
LIN {X 0,Y 274.132,Z 417.121,A -85,B 0,C 180,E1 -20203.579,E2 -20203.579} C_VEL
LIN {X 0,Y 275.68,Z 421.301,A -85,B 0,C 180,E1 -20206.358,E2 -20206.358} C_VEL
LIN {X 0,Y 275.925,Z 422.454,A -85,B 0,C 180,E1 -20206.772,E2 -20206.772} C_VEL
LIN {X 0,Y 275.886,Z 424.336,A -85,B 0,C 180,E1 -20207.094,E2 -20207.094} C_VEL
LIN {X 0,Y 274.12,Z 441.496,A -85,B 0,C 180,E1 -20208.762,E2 -20208.762} C_VEL
LIN {X 0,Y 272.31,Z 458.855,A -85,B 0,C 180,E1 -20210.218,E2 -20210.218} C_VEL
LIN {X 0,Y 271.239,Z 467.752,A -85,B 0,C 180,E1 -20210.799,E2 -20210.799} C_VEL
LIN {X 0,Y 268.058,Z 485.177,A -85,B 0,C 180,E1 -20211.607,E2 -20211.607} C_VEL
LIN {X 0,Y 264.128,Z 500.074,A -85,B 0,C 180,E1 -20212.506,E2 -20212.506} C_VEL
LIN {X 0,Y 259.992,Z 512.773,A -85,B 0,C 180,E1 -20213.508,E2 -20213.508} C_VEL
LIN {X 0,Y 254.845,Z 525.897,A -85,B 0,C 180,E1 -20214.852,E2 -20214.852} C_VEL
LIN {X 0,Y 249.488,Z 537.706,A -85,B 0,C 180,E1 -20216.438,E2 -20216.438} C_VEL
LIN {X 0,Y 244.053,Z 548.53,A -85,B 0,C 180,E1 -20218.294,E2 -20218.294} C_VEL
LIN {X 0,Y 238.707,Z 558.208,A -85,B 0,C 180,E1 -20220.451,E2 -20220.451} C_VEL
LIN {X 0,Y 234.215,Z 566.279,A -85,B 0,C 180,E1 -20222.767,E2 -20222.767} C_VEL
LIN {X 0,Y 229.428,Z 574.04,A -85,B 0,C 180,E1 -20225.572,E2 -20225.572} C_VEL
LIN {X 0,Y 226.069,Z 579.459,A -85,B 0,C 180,E1 -20228.095,E2 -20228.095} C_VEL
LIN {X 0,Y 223.618,Z 583.545,A -85,B 0,C 180,E1 -20230.54,E2 -20230.54} C_VEL
LIN {X 0,Y 221.502,Z 587.253,A -85,B 0,C 180,E1 -20233.407,E2 -20233.407} C_VEL
LIN {X 0,Y 219.842,Z 590.497,A -85,B 0,C 180,E1 -20237.069,E2 -20237.069} C_VEL
LIN {X 0,Y 219.356,Z 592.177,A -85,B 0,C 180,E1 -20240.781,E2 -20240.781} C_VEL
LIN {X 0,Y 219.892,Z 592.36,A -85,B 0,C 180,E1 -20244.497,E2 -20244.497} C_VEL
LIN {X 0,Y 220.292,Z 591.822,A -85,B 0,C 180,E1 -20246.341,E2 -20246.341} C_VEL
LIN {X 0,Y 220.842,Z 590.825,A -85,B 0,C 180,E1 -20248.176,E2 -20248.176} C_VEL
LIN {X 0,Y 221.521,Z 589.183,A -85,B 0,C 180,E1 -20250.341,E2 -20250.341} C_VEL
LIN {X 0,Y 221.038,Z 590.502,A -85,B 0,C 180,E1 -20251.822,E2 -20251.822} C_VEL
LIN {X 0,Y 220.479,Z 591.694,A -85,B 0,C 180,E1 -20253.655,E2 -20253.655} C_VEL
LIN {X 0,Y 219.642,Z 592.766,A -85,B 0,C 180,E1 -20257.28,E2 -20257.28} C_VEL
LIN {X 0,Y 219.513,Z 592.315,A -85,B 0,C 180,E1 -20261.075,E2 -20261.075} C_VEL
LIN {X 0,Y 220.566,Z 590.407,A -85,B 0,C 180,E1 -20264.768,E2 -20264.768} C_VEL
LIN {X 0,Y 222.805,Z 587.008,A -85,B 0,C 180,E1 -20268.387,E2 -20268.387} C_VEL
LIN {X 0,Y 225.22,Z 583.51,A -85,B 0,C 180,E1 -20271.03,E2 -20271.03} C_VEL
LIN {X 0,Y 228.343,Z 579.107,A -85,B 0,C 180,E1 -20273.585,E2 -20273.585} C_VEL
LIN {X 0,Y 232.875,Z 572.718,A -85,B 0,C 180,E1 -20276.432,E2 -20276.432} C_VEL
LIN {X 0,Y 238.212,Z 564.846,A -85,B 0,C 180,E1 -20279.13,E2 -20279.13} C_VEL
LIN {X 0,Y 244.331,Z 555.278,A -85,B 0,C 180,E1 -20281.665,E2 -20281.665} C_VEL
LIN {X 0,Y 250.272,Z 545.306,A -85,B 0,C 180,E1 -20283.684,E2 -20283.684} C_VEL
LIN {X 0,Y 256.861,Z 533.313,A -85,B 0,C 180,E1 -20285.551,E2 -20285.551} C_VEL
LIN {X 0,Y 263.263,Z 519.919,A -85,B 0,C 180,E1 -20287.156,E2 -20287.156} C_VEL
LIN {X 0,Y 268.584,Z 507.308,A -85,B 0,C 180,E1 -20288.278,E2 -20288.278} C_VEL
LIN {X 0,Y 273.493,Z 493.489,A -85,B 0,C 180,E1 -20289.24,E2 -20289.24} C_VEL
LIN {X 0,Y 278.069,Z 477.005,A -85,B 0,C 180,E1 -20290.126,E2 -20290.126} C_VEL
LIN {X 0,Y 280.552,Z 464.774,A -85,B 0,C 180,E1 -20290.738,E2 -20290.738} C_VEL
LIN {X 0,Y 282.176,Z 453.927,A -85,B 0,C 180,E1 -20291.705,E2 -20291.705} C_VEL
LIN {X 0,Y 283.649,Z 443.499,A -85,B 0,C 180,E1 -20292.893,E2 -20292.893} C_VEL
LIN {X 0,Y 283.443,Z 437.989,A -85,B 0,C 180,E1 -20295.318,E2 -20295.318} C_VEL
LIN {X 0,Y 283.646,Z 435.412,A -85,B 0,C 180,E1 -20297.43,E2 -20297.43} C_VEL
LIN {X 0,Y 284.134,Z 434.304,A -85,B 0,C 180,E1 -20298.898,E2 -20298.898} C_VEL
LIN {X 0,Y 286.005,Z 434.564,A -85,B 0,C 180,E1 -20302.048,E2 -20302.048} C_VEL
LIN {X 0,Y 280.772,Z 460.164,A -85,B 0,C 180,E1 -20303.468,E2 -20303.468} C_VEL
LIN {X 0,Y 277.642,Z 472.662,A -85,B 0,C 180,E1 -20304.394,E2 -20304.394} C_VEL
LIN {X 0,Y 273.647,Z 485.236,A -85,B 0,C 180,E1 -20305.596,E2 -20305.596} C_VEL
LIN {X 0,Y 268.693,Z 497.73,A -85,B 0,C 180,E1 -20307.129,E2 -20307.129} C_VEL
LIN {X 0,Y 262.952,Z 509.686,A -85,B 0,C 180,E1 -20309.035,E2 -20309.035} C_VEL
LIN {X 0,Y 257.475,Z 519.324,A -85,B 0,C 180,E1 -20311.019,E2 -20311.019} C_VEL
LIN {X 0,Y 252.273,Z 527.225,A -85,B 0,C 180,E1 -20313.082,E2 -20313.082} C_VEL
LIN {X 0,Y 246.664,Z 534.57,A -85,B 0,C 180,E1 -20315.597,E2 -20315.597} C_VEL
LIN {X 0,Y 242.245,Z 539.538,A -85,B 0,C 180,E1 -20317.842,E2 -20317.842} C_VEL
LIN {X 0,Y 238.158,Z 543.431,A -85,B 0,C 180,E1 -20320.161,E2 -20320.161} C_VEL
LIN {X 0,Y 234.496,Z 546.305,A -85,B 0,C 180,E1 -20322.559,E2 -20322.559} C_VEL
LIN {X 0,Y 230.18,Z 548.711,A -85,B 0,C 180,E1 -20325.861,E2 -20325.861} C_VEL
LIN {X 0,Y 228.344,Z 549.279,A -85,B 0,C 180,E1 -20327.557,E2 -20327.557} C_VEL
LIN {X 0,Y 225.244,Z 549.219,A -85,B 0,C 180,E1 -20331.024,E2 -20331.024} C_VEL
LIN {X 0,Y 223.976,Z 548.611,A -85,B 0,C 180,E1 -20332.789,E2 -20332.789} C_VEL
LIN {X 0,Y 222.85,Z 547.582,A -85,B 0,C 180,E1 -20334.57,E2 -20334.57} C_VEL
LIN {X 0,Y 222.019,Z 546.126,A -85,B 0,C 180,E1 -20336.369,E2 -20336.369} C_VEL
LIN {X 0,Y 221.003,Z 543.189,A -85,B 0,C 180,E1 -20339.088,E2 -20339.088} C_VEL
LIN {X 0,Y 220.25,Z 539.245,A -85,B 0,C 180,E1 -20341.828,E2 -20341.828} C_VEL
LIN {X 0,Y 220.07,Z 534.21,A -85,B 0,C 180,E1 -20344.578,E2 -20344.578} C_VEL
LIN {X 0,Y 220.232,Z 527.948,A -85,B 0,C 180,E1 -20347.333,E2 -20347.333} C_VEL
LIN {X 0,Y 220.628,Z 520.273,A -85,B 0,C 180,E1 -20350.089,E2 -20350.089} C_VEL
LIN {X 0,Y 221.14,Z 510.742,A -85,B 0,C 180,E1 -20352.853,E2 -20352.853} C_VEL
LIN {X 0,Y 221.986,Z 500.094,A -85,B 0,C 180,E1 -20355.375,E2 -20355.375} C_VEL
LIN {X 0,Y 222.832,Z 489.372,A -85,B 0,C 180,E1 -20357.434,E2 -20357.434} C_VEL
LIN {X 0,Y 223.744,Z 476.465,A -85,B 0,C 180,E1 -20359.445,E2 -20359.445} C_VEL
LIN {X 0,Y 224.66,Z 462.935,A -85,B 0,C 180,E1 -20361.084,E2 -20361.084} C_VEL
LIN {X 0,Y 225.399,Z 449.412,A -85,B 0,C 180,E1 -20362.333,E2 -20362.333} C_VEL
LIN {X 0,Y 225.955,Z 434.642,A -85,B 0,C 180,E1 -20363.302,E2 -20363.302} C_VEL
LIN {X 0,Y 227.907,Z 380.033,A -85,B 0,C 180,E1 -20366.104,E2 -20366.104} C_VEL
LIN {X 0,Y 227.683,Z 377.93,A -85,B 0,C 180,E1 -20366.223,E2 -20366.223} C_VEL
LIN {X 0,Y 220.914,Z 353.964,A -85,B 0,C 180,E1 -20367.827,E2 -20367.827} C_VEL
LIN {X 0,Y 220.862,Z 353.971,A -85,B 0,C 180,E1 -20370.778,E2 -20370.778} C_VEL
LIN {X 0,Y 220.8,Z 353.982,A -85,B 0,C 180,E1 -20374.954,E2 -20374.954} C_VEL
LIN {X 0,Y 220.805,Z 353.977,A -85,B 0,C 180,E1 -20379.536,E2 -20379.536} C_VEL
LIN {X 0,Y 220.774,Z 353.984,A -85,B 0,C 180,E1 -20384.453,E2 -20384.453} C_VEL
LIN {X 0,Y 220.774,Z 353.98,A -85,B 0,C 180,E1 -20388.048,E2 -20388.048} C_VEL
LIN {X 0,Y 220.83,Z 353.978,A -85,B 0,C 180,E1 -20392.794,E2 -20392.794} C_VEL
LIN {X 0,Y 220.82,Z 353.976,A -85,B 0,C 180,E1 -20397.245,E2 -20397.245} C_VEL
LIN {X 0,Y 220.824,Z 353.976,A -85,B 0,C 180,E1 -20401.485,E2 -20401.485} C_VEL
LIN {X 0,Y 220.865,Z 353.969,A -85,B 0,C 180,E1 -20405.565,E2 -20405.565} C_VEL
LIN {X 0,Y 220.89,Z 353.968,A -85,B 0,C 180,E1 -20409.514,E2 -20409.514} C_VEL
LIN {X 0,Y 221.014,Z 353.95,A -85,B 0,C 180,E1 -20413.37,E2 -20413.37} C_VEL
LIN {X 0,Y 221.114,Z 353.94,A -85,B 0,C 180,E1 -20419.006,E2 -20419.006} C_VEL
LIN {X 0,Y 221.309,Z 353.917,A -85,B 0,C 180,E1 -20422.702,E2 -20422.702} C_VEL
LIN {X 0,Y 221.511,Z 353.892,A -85,B 0,C 180,E1 -20428.182,E2 -20428.182} C_VEL
LIN {X 0,Y 221.511,Z 353.89,A -85,B 0,C 180,E1 -20431.818,E2 -20431.818} C_VEL
LIN {X 0,Y 221.309,Z 353.914,A -85,B 0,C 180,E1 -20437.298,E2 -20437.298} C_VEL
LIN {X 0,Y 221.115,Z 353.94,A -85,B 0,C 180,E1 -20440.994,E2 -20440.994} C_VEL
LIN {X 0,Y 221.015,Z 353.951,A -85,B 0,C 180,E1 -20446.63,E2 -20446.63} C_VEL
LIN {X 0,Y 220.891,Z 353.97,A -85,B 0,C 180,E1 -20450.487,E2 -20450.487} C_VEL
LIN {X 0,Y 220.866,Z 353.97,A -85,B 0,C 180,E1 -20454.436,E2 -20454.436} C_VEL
LIN {X 0,Y 220.826,Z 353.978,A -85,B 0,C 180,E1 -20458.516,E2 -20458.516} C_VEL
LIN {X 0,Y 220.822,Z 353.975,A -85,B 0,C 180,E1 -20462.756,E2 -20462.756} C_VEL
LIN {X 0,Y 220.837,Z 353.974,A -85,B 0,C 180,E1 -20467.289,E2 -20467.289} C_VEL
LIN {X 0,Y 220.774,Z 353.983,A -85,B 0,C 180,E1 -20471.952,E2 -20471.952} C_VEL
LIN {X 0,Y 220.773,Z 353.983,A -85,B 0,C 180,E1 -20475.547,E2 -20475.547} C_VEL
LIN {X 0,Y 220.807,Z 353.976,A -85,B 0,C 180,E1 -20480.464,E2 -20480.464} C_VEL
LIN {X 0,Y 220.936,Z 353.963,A -85,B 0,C 180,E1 -20485.401,E2 -20485.401} C_VEL
LIN {X 0,Y 226.882,Z 373.871,A -85,B 0,C 180,E1 -20486.759,E2 -20486.759} C_VEL
LIN {X 0,Y 228.847,Z 380.918,A -85,B 0,C 180,E1 -20487.2,E2 -20487.2} C_VEL
LIN {X 0,Y 226.781,Z 433.077,A -85,B 0,C 180,E1 -20489.699,E2 -20489.699} C_VEL
LIN {X 0,Y 226.297,Z 447.561,A -85,B 0,C 180,E1 -20490.574,E2 -20490.574} C_VEL
LIN {X 0,Y 225.476,Z 462.244,A -85,B 0,C 180,E1 -20491.873,E2 -20491.873} C_VEL
LIN {X 0,Y 224.635,Z 474.192,A -85,B 0,C 180,E1 -20493.274,E2 -20493.274} C_VEL
LIN {X 0,Y 223.612,Z 486.796,A -85,B 0,C 180,E1 -20495.143,E2 -20495.143} C_VEL
LIN {X 0,Y 222.588,Z 498.115,A -85,B 0,C 180,E1 -20497.25,E2 -20497.25} C_VEL
LIN {X 0,Y 221.679,Z 508.39,A -85,B 0,C 180,E1 -20499.591,E2 -20499.591} C_VEL
LIN {X 0,Y 220.925,Z 517.912,A -85,B 0,C 180,E1 -20502.285,E2 -20502.285} C_VEL
LIN {X 0,Y 220.409,Z 526.29,A -85,B 0,C 180,E1 -20505.222,E2 -20505.222} C_VEL
LIN {X 0,Y 220.171,Z 532.668,A -85,B 0,C 180,E1 -20508.026,E2 -20508.026} C_VEL
LIN {X 0,Y 220.416,Z 538.504,A -85,B 0,C 180,E1 -20511.284,E2 -20511.284} C_VEL
LIN {X 0,Y 220.861,Z 542.784,A -85,B 0,C 180,E1 -20514.523,E2 -20514.523} C_VEL
LIN {X 0,Y 222.129,Z 545.964,A -85,B 0,C 180,E1 -20518.188,E2 -20518.188} C_VEL
LIN {X 0,Y 223.05,Z 546.918,A -85,B 0,C 180,E1 -20520.001,E2 -20520.001} C_VEL
LIN {X 0,Y 225.311,Z 547.558,A -85,B 0,C 180,E1 -20523.468,E2 -20523.468} C_VEL
LIN {X 0,Y 226.781,Z 547.293,A -85,B 0,C 180,E1 -20525.335,E2 -20525.335} C_VEL
LIN {X 0,Y 228.475,Z 546.561,A -85,B 0,C 180,E1 -20527.069,E2 -20527.069} C_VEL
LIN {X 0,Y 232.284,Z 543.904,A -85,B 0,C 180,E1 -20530.46,E2 -20530.46} C_VEL
LIN {X 0,Y 235.598,Z 540.745,A -85,B 0,C 180,E1 -20532.929,E2 -20532.929} C_VEL
LIN {X 0,Y 239.312,Z 536.54,A -85,B 0,C 180,E1 -20535.327,E2 -20535.327} C_VEL
LIN {X 0,Y 243.491,Z 530.922,A -85,B 0,C 180,E1 -20537.729,E2 -20537.729} C_VEL
LIN {X 0,Y 247.785,Z 524.426,A -85,B 0,C 180,E1 -20539.9,E2 -20539.9} C_VEL
LIN {X 0,Y 252.601,Z 516.099,A -85,B 0,C 180,E1 -20542.062,E2 -20542.062} C_VEL
LIN {X 0,Y 256.728,Z 507.739,A -85,B 0,C 180,E1 -20543.816,E2 -20543.816} C_VEL
LIN {X 0,Y 261.108,Z 497.574,A -85,B 0,C 180,E1 -20545.51,E2 -20545.51} C_VEL
LIN {X 0,Y 264.692,Z 487.719,A -85,B 0,C 180,E1 -20546.833,E2 -20546.833} C_VEL
LIN {X 0,Y 268.291,Z 475.747,A -85,B 0,C 180,E1 -20548.134,E2 -20548.134} C_VEL
LIN {X 0,Y 271.33,Z 462.735,A -85,B 0,C 180,E1 -20549.216,E2 -20549.216} C_VEL
LIN {X 0,Y 273.614,Z 449.18,A -85,B 0,C 180,E1 -20550.062,E2 -20550.062} C_VEL
LIN {X 0,Y 277.257,Z 427.316,A -85,B 0,C 180,E1 -20551.115,E2 -20551.115} C_VEL
LIN {X 0,Y 277.368,Z 425.436,A -85,B 0,C 180,E1 -20551.352,E2 -20551.352} C_VEL
LIN {X 0,Y 277.079,Z 424.228,A -85,B 0,C 180,E1 -20551.761,E2 -20551.761} C_VEL
LIN {X 0,Y 276.071,Z 423.394,A -85,B 0,C 180,E1 -20552.658,E2 -20552.658} C_VEL
LIN {X 0,Y 273.415,Z 423.889,A -85,B 0,C 180,E1 -20554.903,E2 -20554.903} C_VEL
LIN {X 0,Y 273.055,Z 423.588,A -85,B 0,C 180,E1 -20555.394,E2 -20555.394} C_VEL
LIN {X 0,Y 272.241,Z 421.556,A -85,B 0,C 180,E1 -20557.615,E2 -20557.615} C_VEL
LIN {X 0,Y 271.749,Z 421.735,A -85,B 0,C 180,E1 -20559.996,E2 -20559.996} C_VEL
LIN {X 0,Y 272.378,Z 424.005,A -85,B 0,C 180,E1 -20563.411,E2 -20563.411} C_VEL
LIN {X 0,Y 273.578,Z 427.667,A -85,B 0,C 180,E1 -20565.872,E2 -20565.872} C_VEL
LIN {X 0,Y 271.507,Z 444.459,A -85,B 0,C 180,E1 -20567.514,E2 -20567.514} C_VEL
LIN {X 0,Y 269.583,Z 460.497,A -85,B 0,C 180,E1 -20568.88,E2 -20568.88} C_VEL
LIN {X 0,Y 268.457,Z 468.72,A -85,B 0,C 180,E1 -20569.43,E2 -20569.43} C_VEL
LIN {X 0,Y 265.176,Z 484.927,A -85,B 0,C 180,E1 -20570.199,E2 -20570.199} C_VEL
LIN {X 0,Y 260.631,Z 500.946,A -85,B 0,C 180,E1 -20571.174,E2 -20571.174} C_VEL
LIN {X 0,Y 256.296,Z 513.077,A -85,B 0,C 180,E1 -20572.152,E2 -20572.152} C_VEL
LIN {X 0,Y 250.946,Z 525.743,A -85,B 0,C 180,E1 -20573.478,E2 -20573.478} C_VEL
LIN {X 0,Y 245.322,Z 537.359,A -85,B 0,C 180,E1 -20575.042,E2 -20575.042} C_VEL
LIN {X 0,Y 240.126,Z 547.013,A -85,B 0,C 180,E1 -20576.716,E2 -20576.716} C_VEL
LIN {X 0,Y 234.43,Z 556.728,A -85,B 0,C 180,E1 -20578.859,E2 -20578.859} C_VEL
LIN {X 0,Y 229.453,Z 564.771,A -85,B 0,C 180,E1 -20581.156,E2 -20581.156} C_VEL
LIN {X 0,Y 224.349,Z 572.551,A -85,B 0,C 180,E1 -20583.987,E2 -20583.987} C_VEL
LIN {X 0,Y 220.599,Z 577.962,A -85,B 0,C 180,E1 -20586.532,E2 -20586.532} C_VEL
LIN {X 0,Y 217.596,Z 582.361,A -85,B 0,C 180,E1 -20589.189,E2 -20589.189} C_VEL
LIN {X 0,Y 215.341,Z 585.842,A -85,B 0,C 180,E1 -20591.937,E2 -20591.937} C_VEL
LIN {X 0,Y 213.647,Z 588.457,A -85,B 0,C 180,E1 -20594.742,E2 -20594.742} C_VEL
LIN {X 0,Y 212.468,Z 590.63,A -85,B 0,C 180,E1 -20598.552,E2 -20598.552} C_VEL
LIN {X 0,Y 212.475,Z 591.333,A -85,B 0,C 180,E1 -20602.397,E2 -20602.397} C_VEL
LIN {X 0,Y 212.865,Z 591.082,A -85,B 0,C 180,E1 -20604.315,E2 -20604.315} C_VEL
LIN {X 0,Y 213.318,Z 590.417,A -85,B 0,C 180,E1 -20606.222,E2 -20606.222} C_VEL
LIN {X 0,Y 213.9,Z 589.345,A -85,B 0,C 180,E1 -20608.117,E2 -20608.117} C_VEL
LIN {X 0,Y 214.636,Z 587.478,A -85,B 0,C 180,E1 -20610.469,E2 -20610.469} C_VEL
LIN {X 0,Y 213.523,Z 590.091,A -85,B 0,C 180,E1 -20613.774,E2 -20613.774} C_VEL
LIN {X 0,Y 212.621,Z 591.462,A -85,B 0,C 180,E1 -20617.597,E2 -20617.597} C_VEL
LIN {X 0,Y 212.54,Z 591.261,A -85,B 0,C 180,E1 -20621.443,E2 -20621.443} C_VEL
LIN {X 0,Y 213.673,Z 589.638,A -85,B 0,C 180,E1 -20625.256,E2 -20625.256} C_VEL
LIN {X 0,Y 216.025,Z 586.619,A -85,B 0,C 180,E1 -20628.986,E2 -20628.986} C_VEL
LIN {X 0,Y 218.586,Z 583.383,A -85,B 0,C 180,E1 -20631.7,E2 -20631.7} C_VEL
LIN {X 0,Y 221.871,Z 579.301,A -85,B 0,C 180,E1 -20634.317,E2 -20634.317} C_VEL
LIN {X 0,Y 225.856,Z 574.303,A -85,B 0,C 180,E1 -20636.82,E2 -20636.82} C_VEL
LIN {X 0,Y 231.27,Z 567.155,A -85,B 0,C 180,E1 -20639.592,E2 -20639.592} C_VEL
LIN {X 0,Y 237.47,Z 558.466,A -85,B 0,C 180,E1 -20642.189,E2 -20642.189} C_VEL
LIN {X 0,Y 243.472,Z 549.498,A -85,B 0,C 180,E1 -20644.255,E2 -20644.255} C_VEL
LIN {X 0,Y 250.101,Z 538.727,A -85,B 0,C 180,E1 -20646.165,E2 -20646.165} C_VEL
LIN {X 0,Y 256.687,Z 526.896,A -85,B 0,C 180,E1 -20647.779,E2 -20647.779} C_VEL
LIN {X 0,Y 261.771,Z 516.483,A -85,B 0,C 180,E1 -20648.926,E2 -20648.926} C_VEL
LIN {X 0,Y 268.012,Z 502.042,A -85,B 0,C 180,E1 -20650.092,E2 -20650.092} C_VEL
LIN {X 0,Y 273.275,Z 486.929,A -85,B 0,C 180,E1 -20651.042,E2 -20651.042} C_VEL
LIN {X 0,Y 277.467,Z 471.217,A -85,B 0,C 180,E1 -20651.824,E2 -20651.824} C_VEL
LIN {X 0,Y 278.639,Z 465.495,A -85,B 0,C 180,E1 -20652.168,E2 -20652.168} C_VEL
LIN {X 0,Y 280.249,Z 456.058,A -85,B 0,C 180,E1 -20653.038,E2 -20653.038} C_VEL
LIN {X 0,Y 281.49,Z 448.592,A -85,B 0,C 180,E1 -20653.904,E2 -20653.904} C_VEL
LIN {X 0,Y 281.577,Z 444.358,A -85,B 0,C 180,E1 -20655.866,E2 -20655.866} C_VEL
LIN {X 0,Y 281.902,Z 442.164,A -85,B 0,C 180,E1 -20657.69,E2 -20657.69} C_VEL
LIN {X 0,Y 282.348,Z 441.22,A -85,B 0,C 180,E1 -20658.924,E2 -20658.924} C_VEL
LIN {X 0,Y 283.378,Z 441.216,A -85,B 0,C 180,E1 -20660.968,E2 -20660.968} C_VEL
LIN {X 0,Y 278.912,Z 461.616,A -85,B 0,C 180,E1 -20662.096,E2 -20662.096} C_VEL
LIN {X 0,Y 275.657,Z 473.807,A -85,B 0,C 180,E1 -20662.991,E2 -20662.991} C_VEL
LIN {X 0,Y 270.965,Z 487.464,A -85,B 0,C 180,E1 -20664.296,E2 -20664.296} C_VEL
LIN {X 0,Y 265.488,Z 500.216,A -85,B 0,C 180,E1 -20665.883,E2 -20665.883} C_VEL
LIN {X 0,Y 259.682,Z 511.395,A -85,B 0,C 180,E1 -20667.688,E2 -20667.688} C_VEL
LIN {X 0,Y 253.849,Z 520.9,A -85,B 0,C 180,E1 -20669.65,E2 -20669.65} C_VEL
LIN {X 0,Y 248.343,Z 528.676,A -85,B 0,C 180,E1 -20671.704,E2 -20671.704} C_VEL
LIN {X 0,Y 242.34,Z 535.94,A -85,B 0,C 180,E1 -20674.213,E2 -20674.213} C_VEL
LIN {X 0,Y 237.95,Z 540.52,A -85,B 0,C 180,E1 -20676.292,E2 -20676.292} C_VEL
LIN {X 0,Y 233.183,Z 544.708,A -85,B 0,C 180,E1 -20678.796,E2 -20678.796} C_VEL
LIN {X 0,Y 230.498,Z 546.722,A -85,B 0,C 180,E1 -20680.403,E2 -20680.403} C_VEL
LIN {X 0,Y 228.003,Z 548.317,A -85,B 0,C 180,E1 -20682.046,E2 -20682.046} C_VEL
LIN {X 0,Y 223.477,Z 550.251,A -85,B 0,C 180,E1 -20685.428,E2 -20685.428} C_VEL
LIN {X 0,Y 219.803,Z 550.629,A -85,B 0,C 180,E1 -20688.939,E2 -20688.939} C_VEL
LIN {X 0,Y 216.988,Z 549.363,A -85,B 0,C 180,E1 -20692.555,E2 -20692.555} C_VEL
LIN {X 0,Y 214.94,Z 546.543,A -85,B 0,C 180,E1 -20696.25,E2 -20696.25} C_VEL
LIN {X 0,Y 213.891,Z 543.31,A -85,B 0,C 180,E1 -20699.058,E2 -20699.058} C_VEL
LIN {X 0,Y 213.161,Z 539.07,A -85,B 0,C 180,E1 -20701.889,E2 -20701.889} C_VEL
LIN {X 0,Y 213.033,Z 532.686,A -85,B 0,C 180,E1 -20705.204,E2 -20705.204} C_VEL
LIN {X 0,Y 213.138,Z 527.091,A -85,B 0,C 180,E1 -20707.578,E2 -20707.578} C_VEL
LIN {X 0,Y 213.594,Z 518.956,A -85,B 0,C 180,E1 -20710.425,E2 -20710.425} C_VEL
LIN {X 0,Y 214.18,Z 508.968,A -85,B 0,C 180,E1 -20713.278,E2 -20713.278} C_VEL
LIN {X 0,Y 215.092,Z 497.647,A -85,B 0,C 180,E1 -20715.881,E2 -20715.881} C_VEL
LIN {X 0,Y 215.906,Z 486.197,A -85,B 0,C 180,E1 -20718.012,E2 -20718.012} C_VEL
LIN {X 0,Y 216.911,Z 472.776,A -85,B 0,C 180,E1 -20720.014,E2 -20720.014} C_VEL
LIN {X 0,Y 217.756,Z 459.564,A -85,B 0,C 180,E1 -20721.537,E2 -20721.537} C_VEL
LIN {X 0,Y 218.536,Z 445.372,A -85,B 0,C 180,E1 -20722.762,E2 -20722.762} C_VEL
LIN {X 0,Y 219.115,Z 423.953,A -85,B 0,C 180,E1 -20724.012,E2 -20724.012} C_VEL
LIN {X 0,Y 220.849,Z 379.788,A -85,B 0,C 180,E1 -20726.382,E2 -20726.382} C_VEL
LIN {X 0,Y 213.858,Z 354.843,A -85,B 0,C 180,E1 -20728.065,E2 -20728.065} C_VEL
LIN {X 0,Y 213.776,Z 354.853,A -85,B 0,C 180,E1 -20731.735,E2 -20731.735} C_VEL
LIN {X 0,Y 213.742,Z 354.859,A -85,B 0,C 180,E1 -20736.287,E2 -20736.287} C_VEL
LIN {X 0,Y 213.711,Z 354.864,A -85,B 0,C 180,E1 -20741.124,E2 -20741.124} C_VEL
LIN {X 0,Y 213.706,Z 354.863,A -85,B 0,C 180,E1 -20743.677,E2 -20743.677} C_VEL
LIN {X 0,Y 213.707,Z 354.862,A -85,B 0,C 180,E1 -20746.342,E2 -20746.342} C_VEL
LIN {X 0,Y 213.734,Z 354.86,A -85,B 0,C 180,E1 -20751.336,E2 -20751.336} C_VEL
LIN {X 0,Y 213.766,Z 354.852,A -85,B 0,C 180,E1 -20756.02,E2 -20756.02} C_VEL
LIN {X 0,Y 213.758,Z 354.859,A -85,B 0,C 180,E1 -20760.451,E2 -20760.451} C_VEL
LIN {X 0,Y 213.799,Z 354.852,A -85,B 0,C 180,E1 -20764.702,E2 -20764.702} C_VEL
LIN {X 0,Y 213.811,Z 354.852,A -85,B 0,C 180,E1 -20768.803,E2 -20768.803} C_VEL
LIN {X 0,Y 213.941,Z 354.833,A -85,B 0,C 180,E1 -20772.804,E2 -20772.804} C_VEL
LIN {X 0,Y 213.978,Z 354.832,A -85,B 0,C 180,E1 -20776.708,E2 -20776.708} C_VEL
LIN {X 0,Y 214.194,Z 354.801,A -85,B 0,C 180,E1 -20780.558,E2 -20780.558} C_VEL
LIN {X 0,Y 214.246,Z 354.796,A -85,B 0,C 180,E1 -20782.461,E2 -20782.461} C_VEL
LIN {X 0,Y 214.444,Z 354.772,A -85,B 0,C 180,E1 -20788.122,E2 -20788.122} C_VEL
LIN {X 0,Y 214.548,Z 354.756,A -85,B 0,C 180,E1 -20790,E2 -20790} C_VEL
LIN {X 0,Y 214.444,Z 354.77,A -85,B 0,C 180,E1 -20791.878,E2 -20791.878} C_VEL
LIN {X 0,Y 214.246,Z 354.794,A -85,B 0,C 180,E1 -20797.54,E2 -20797.54} C_VEL
LIN {X 0,Y 214.046,Z 354.82,A -85,B 0,C 180,E1 -20801.362,E2 -20801.362} C_VEL
LIN {X 0,Y 213.932,Z 354.833,A -85,B 0,C 180,E1 -20805.237,E2 -20805.237} C_VEL
LIN {X 0,Y 213.838,Z 354.846,A -85,B 0,C 180,E1 -20809.188,E2 -20809.188} C_VEL
LIN {X 0,Y 213.846,Z 354.845,A -85,B 0,C 180,E1 -20813.228,E2 -20813.228} C_VEL
LIN {X 0,Y 213.828,Z 354.847,A -85,B 0,C 180,E1 -20817.451,E2 -20817.451} C_VEL
LIN {X 0,Y 213.769,Z 354.856,A -85,B 0,C 180,E1 -20821.738,E2 -20821.738} C_VEL
LIN {X 0,Y 213.751,Z 354.86,A -85,B 0,C 180,E1 -20826.287,E2 -20826.287} C_VEL
LIN {X 0,Y 213.715,Z 354.86,A -85,B 0,C 180,E1 -20831.125,E2 -20831.125} C_VEL
LIN {X 0,Y 213.707,Z 354.861,A -85,B 0,C 180,E1 -20833.679,E2 -20833.679} C_VEL
LIN {X 0,Y 213.706,Z 354.865,A -85,B 0,C 180,E1 -20836.345,E2 -20836.345} C_VEL
LIN {X 0,Y 213.734,Z 354.856,A -85,B 0,C 180,E1 -20841.337,E2 -20841.337} C_VEL
LIN {X 0,Y 213.877,Z 354.909,A -85,B 0,C 180,E1 -20845.091,E2 -20845.091} C_VEL
LIN {X 0,Y 221.835,Z 381.842,A -85,B 0,C 180,E1 -20846.923,E2 -20846.923} C_VEL
LIN {X 0,Y 219.755,Z 433.879,A -85,B 0,C 180,E1 -20849.517,E2 -20849.517} C_VEL
LIN {X 0,Y 219.221,Z 448.441,A -85,B 0,C 180,E1 -20850.427,E2 -20850.427} C_VEL
LIN {X 0,Y 218.347,Z 463.322,A -85,B 0,C 180,E1 -20851.788,E2 -20851.788} C_VEL
LIN {X 0,Y 217.405,Z 476.073,A -85,B 0,C 180,E1 -20853.351,E2 -20853.351} C_VEL
LIN {X 0,Y 216.415,Z 488.417,A -85,B 0,C 180,E1 -20855.273,E2 -20855.273} C_VEL
LIN {X 0,Y 215.311,Z 500.685,A -85,B 0,C 180,E1 -20857.701,E2 -20857.701} C_VEL
LIN {X 0,Y 214.469,Z 509.689,A -85,B 0,C 180,E1 -20859.876,E2 -20859.876} C_VEL
LIN {X 0,Y 213.808,Z 518.372,A -85,B 0,C 180,E1 -20862.413,E2 -20862.413} C_VEL
LIN {X 0,Y 213.309,Z 526.243,A -85,B 0,C 180,E1 -20865.207,E2 -20865.207} C_VEL
LIN {X 0,Y 213.087,Z 531.856,A -85,B 0,C 180,E1 -20867.622,E2 -20867.622} C_VEL
LIN {X 0,Y 213.21,Z 537.358,A -85,B 0,C 180,E1 -20870.514,E2 -20870.514} C_VEL
LIN {X 0,Y 213.554,Z 541.627,A -85,B 0,C 180,E1 -20873.387,E2 -20873.387} C_VEL
LIN {X 0,Y 214.215,Z 544.841,A -85,B 0,C 180,E1 -20876.239,E2 -20876.239} C_VEL
LIN {X 0,Y 214.983,Z 546.423,A -85,B 0,C 180,E1 -20878.128,E2 -20878.128} C_VEL
LIN {X 0,Y 217.032,Z 548.343,A -85,B 0,C 180,E1 -20881.857,E2 -20881.857} C_VEL
LIN {X 0,Y 218.363,Z 548.687,A -85,B 0,C 180,E1 -20883.692,E2 -20883.692} C_VEL
LIN {X 0,Y 219.8,Z 548.603,A -85,B 0,C 180,E1 -20885.505,E2 -20885.505} C_VEL
LIN {X 0,Y 223.422,Z 547.225,A -85,B 0,C 180,E1 -20889.05,E2 -20889.05} C_VEL
LIN {X 0,Y 225.506,Z 545.901,A -85,B 0,C 180,E1 -20890.778,E2 -20890.778} C_VEL
LIN {X 0,Y 228.933,Z 543.144,A -85,B 0,C 180,E1 -20893.312,E2 -20893.312} C_VEL
LIN {X 0,Y 232.779,Z 539.316,A -85,B 0,C 180,E1 -20895.768,E2 -20895.768} C_VEL
LIN {X 0,Y 237.171,Z 534.226,A -85,B 0,C 180,E1 -20898.218,E2 -20898.218} C_VEL
LIN {X 0,Y 242.441,Z 527.071,A -85,B 0,C 180,E1 -20900.801,E2 -20900.801} C_VEL
LIN {X 0,Y 247.48,Z 519.146,A -85,B 0,C 180,E1 -20902.985,E2 -20902.985} C_VEL
LIN {X 0,Y 251.835,Z 511.184,A -85,B 0,C 180,E1 -20904.748,E2 -20904.748} C_VEL
LIN {X 0,Y 256.436,Z 501.609,A -85,B 0,C 180,E1 -20906.447,E2 -20906.447} C_VEL
LIN {X 0,Y 260.709,Z 491.09,A -85,B 0,C 180,E1 -20907.93,E2 -20907.93} C_VEL
LIN {X 0,Y 264.516,Z 479.681,A -85,B 0,C 180,E1 -20909.224,E2 -20909.224} C_VEL
LIN {X 0,Y 267.848,Z 467.221,A -85,B 0,C 180,E1 -20910.339,E2 -20910.339} C_VEL
LIN {X 0,Y 270.401,Z 454.348,A -85,B 0,C 180,E1 -20911.212,E2 -20911.212} C_VEL
LIN {X 0,Y 274.948,Z 428.306,A -85,B 0,C 180,E1 -20912.505,E2 -20912.505} C_VEL
LIN {X 0,Y 273.743,Z 425.332,A -85,B 0,C 180,E1 -20914.133,E2 -20914.133} C_VEL
LIN {X 0,Y 273.175,Z 423.786,A -85,B 0,C 180,E1 -20915.193,E2 -20915.193} C_VEL
LIN {X 0,Y 273.055,Z 423.588,A -85,B 0,C 180,E1 -20915.394,E2 -20915.394} C_VEL
LIN {X 0,Y 272.559,Z 423.222,A -85,B 0,C 180,E1 -20916.21,E2 -20916.21} C_VEL
LIN {X 0,Y 272.037,Z 423.529,A -85,B 0,C 180,E1 -20917.031,E2 -20917.031} C_VEL
LIN {X 0,Y 271.031,Z 425.435,A -85,B 0,C 180,E1 -20918.65,E2 -20918.65} C_VEL
LIN {X 0,Y 270.18,Z 429.108,A -85,B 0,C 180,E1 -20921.116,E2 -20921.116} C_VEL
LIN {X 0,Y 270.202,Z 429.858,A -85,B 0,C 180,E1 -20921.963,E2 -20921.963} C_VEL
LIN {X 0,Y 270.618,Z 430.987,A -85,B 0,C 180,E1 -20923.284,E2 -20923.284} C_VEL
LIN {X 0,Y 271.237,Z 433.29,A -85,B 0,C 180,E1 -20924.857,E2 -20924.857} C_VEL
LIN {X 0,Y 268.588,Z 451.602,A -85,B 0,C 180,E1 -20926.621,E2 -20926.621} C_VEL
LIN {X 0,Y 266.606,Z 465.588,A -85,B 0,C 180,E1 -20927.746,E2 -20927.746} C_VEL
LIN {X 0,Y 265.615,Z 471.519,A -85,B 0,C 180,E1 -20928.104,E2 -20928.104} C_VEL
LIN {X 0,Y 261.65,Z 488.387,A -85,B 0,C 180,E1 -20928.933,E2 -20928.933} C_VEL
LIN {X 0,Y 256.649,Z 503.839,A -85,B 0,C 180,E1 -20929.944,E2 -20929.944} C_VEL
LIN {X 0,Y 252.165,Z 515.049,A -85,B 0,C 180,E1 -20930.907,E2 -20930.907} C_VEL
LIN {X 0,Y 246.025,Z 528.344,A -85,B 0,C 180,E1 -20932.366,E2 -20932.366} C_VEL
LIN {X 0,Y 240.81,Z 538.171,A -85,B 0,C 180,E1 -20933.772,E2 -20933.772} C_VEL
LIN {X 0,Y 234.344,Z 549.12,A -85,B 0,C 180,E1 -20935.783,E2 -20935.783} C_VEL
LIN {X 0,Y 228.47,Z 558.218,A -85,B 0,C 180,E1 -20937.951,E2 -20937.951} C_VEL
LIN {X 0,Y 223.337,Z 565.777,A -85,B 0,C 180,E1 -20940.289,E2 -20940.289} C_VEL
LIN {X 0,Y 218.024,Z 573.034,A -85,B 0,C 180,E1 -20943.173,E2 -20943.173} C_VEL
LIN {X 0,Y 214.104,Z 578.115,A -85,B 0,C 180,E1 -20945.775,E2 -20945.775} C_VEL
LIN {X 0,Y 210.935,Z 582.227,A -85,B 0,C 180,E1 -20948.5,E2 -20948.5} C_VEL
LIN {X 0,Y 207.875,Z 586.321,A -85,B 0,C 180,E1 -20952.285,E2 -20952.285} C_VEL
LIN {X 0,Y 205.934,Z 588.95,A -85,B 0,C 180,E1 -20956.178,E2 -20956.178} C_VEL
LIN {X 0,Y 205.303,Z 590.075,A -85,B 0,C 180,E1 -20960.144,E2 -20960.144} C_VEL
LIN {X 0,Y 205.838,Z 589.752,A -85,B 0,C 180,E1 -20964.12,E2 -20964.12} C_VEL
LIN {X 0,Y 206.333,Z 588.985,A -85,B 0,C 180,E1 -20966.093,E2 -20966.093} C_VEL
LIN {X 0,Y 206.972,Z 587.777,A -85,B 0,C 180,E1 -20968.054,E2 -20968.054} C_VEL
LIN {X 0,Y 207.806,Z 585.612,A -85,B 0,C 180,E1 -20970.484,E2 -20970.484} C_VEL
LIN {X 0,Y 206.59,Z 588.431,A -85,B 0,C 180,E1 -20973.901,E2 -20973.901} C_VEL
LIN {X 0,Y 205.648,Z 590.025,A -85,B 0,C 180,E1 -20977.857,E2 -20977.857} C_VEL
LIN {X 0,Y 205.582,Z 590.127,A -85,B 0,C 180,E1 -20981.836,E2 -20981.836} C_VEL
LIN {X 0,Y 206.788,Z 588.847,A -85,B 0,C 180,E1 -20985.777,E2 -20985.777} C_VEL
LIN {X 0,Y 209.274,Z 586.157,A -85,B 0,C 180,E1 -20989.623,E2 -20989.623} C_VEL
LIN {X 0,Y 213.045,Z 582.058,A -85,B 0,C 180,E1 -20993.319,E2 -20993.319} C_VEL
LIN {X 0,Y 218.1,Z 576.484,A -85,B 0,C 180,E1 -20996.816,E2 -20996.816} C_VEL
LIN {X 0,Y 222.65,Z 571.203,A -85,B 0,C 180,E1 -20999.292,E2 -20999.292} C_VEL
LIN {X 0,Y 228.768,Z 563.776,A -85,B 0,C 180,E1 -21002.001,E2 -21002.001} C_VEL
LIN {X 0,Y 235.639,Z 554.691,A -85,B 0,C 180,E1 -21004.519,E2 -21004.519} C_VEL
LIN {X 0,Y 242.249,Z 545.329,A -85,B 0,C 180,E1 -21006.494,E2 -21006.494} C_VEL
LIN {X 0,Y 249.405,Z 534.148,A -85,B 0,C 180,E1 -21008.312,E2 -21008.312} C_VEL
LIN {X 0,Y 256.396,Z 521.723,A -85,B 0,C 180,E1 -21009.869,E2 -21009.869} C_VEL
LIN {X 0,Y 262.482,Z 509.531,A -85,B 0,C 180,E1 -21010.995,E2 -21010.995} C_VEL
LIN {X 0,Y 268.802,Z 494.438,A -85,B 0,C 180,E1 -21012.066,E2 -21012.066} C_VEL
LIN {X 0,Y 273.903,Z 479.081,A -85,B 0,C 180,E1 -21012.907,E2 -21012.907} C_VEL
LIN {X 0,Y 276.757,Z 468.014,A -85,B 0,C 180,E1 -21013.479,E2 -21013.479} C_VEL
LIN {X 0,Y 278.61,Z 458.55,A -85,B 0,C 180,E1 -21014.362,E2 -21014.362} C_VEL
LIN {X 0,Y 279.516,Z 453.857,A -85,B 0,C 180,E1 -21014.894,E2 -21014.894} C_VEL
LIN {X 0,Y 279.788,Z 450.757,A -85,B 0,C 180,E1 -21016.387,E2 -21016.387} C_VEL
LIN {X 0,Y 280.196,Z 448.814,A -85,B 0,C 180,E1 -21018.075,E2 -21018.075} C_VEL
LIN {X 0,Y 280.817,Z 447.999,A -85,B 0,C 180,E1 -21019.54,E2 -21019.54} C_VEL
LIN {X 0,Y 280.963,Z 447.977,A -85,B 0,C 180,E1 -21019.858,E2 -21019.858} C_VEL
LIN {X 0,Y 277.329,Z 463.549,A -85,B 0,C 180,E1 -21020.731,E2 -21020.731} C_VEL
LIN {X 0,Y 273.64,Z 476.193,A -85,B 0,C 180,E1 -21021.658,E2 -21021.658} C_VEL
LIN {X 0,Y 269.064,Z 488.609,A -85,B 0,C 180,E1 -21022.84,E2 -21022.84} C_VEL
LIN {X 0,Y 263.546,Z 500.735,A -85,B 0,C 180,E1 -21024.313,E2 -21024.313} C_VEL
LIN {X 0,Y 257.662,Z 511.511,A -85,B 0,C 180,E1 -21026.002,E2 -21026.002} C_VEL
LIN {X 0,Y 252.462,Z 519.71,A -85,B 0,C 180,E1 -21027.596,E2 -21027.596} C_VEL
LIN {X 0,Y 246.659,Z 527.713,A -85,B 0,C 180,E1 -21029.55,E2 -21029.55} C_VEL
LIN {X 0,Y 241.821,Z 533.549,A -85,B 0,C 180,E1 -21031.344,E2 -21031.344} C_VEL
LIN {X 0,Y 236.48,Z 539.171,A -85,B 0,C 180,E1 -21033.525,E2 -21033.525} C_VEL
LIN {X 0,Y 229.962,Z 544.897,A -85,B 0,C 180,E1 -21036.59,E2 -21036.59} C_VEL
LIN {X 0,Y 226.924,Z 547.116,A -85,B 0,C 180,E1 -21038.182,E2 -21038.182} C_VEL
LIN {X 0,Y 221.491,Z 550.212,A -85,B 0,C 180,E1 -21041.499,E2 -21041.499} C_VEL
LIN {X 0,Y 216.765,Z 551.756,A -85,B 0,C 180,E1 -21044.966,E2 -21044.966} C_VEL
LIN {X 0,Y 212.913,Z 551.679,A -85,B 0,C 180,E1 -21048.576,E2 -21048.576} C_VEL
LIN {X 0,Y 210.006,Z 550.061,A -85,B 0,C 180,E1 -21052.306,E2 -21052.306} C_VEL
LIN {X 0,Y 207.856,Z 546.805,A -85,B 0,C 180,E1 -21056.122,E2 -21056.122} C_VEL
LIN {X 0,Y 206.786,Z 543.277,A -85,B 0,C 180,E1 -21059.025,E2 -21059.025} C_VEL
LIN {X 0,Y 206.056,Z 538.718,A -85,B 0,C 180,E1 -21061.954,E2 -21061.954} C_VEL
LIN {X 0,Y 205.968,Z 531.985,A -85,B 0,C 180,E1 -21065.383,E2 -21065.383} C_VEL
LIN {X 0,Y 206.051,Z 526.035,A -85,B 0,C 180,E1 -21067.84,E2 -21067.84} C_VEL
LIN {X 0,Y 206.553,Z 517.474,A -85,B 0,C 180,E1 -21070.785,E2 -21070.785} C_VEL
LIN {X 0,Y 207.236,Z 506.916,A -85,B 0,C 180,E1 -21073.732,E2 -21073.732} C_VEL
LIN {X 0,Y 208.129,Z 496.105,A -85,B 0,C 180,E1 -21076.175,E2 -21076.175} C_VEL
LIN {X 0,Y 208.946,Z 484.133,A -85,B 0,C 180,E1 -21078.38,E2 -21078.38} C_VEL
LIN {X 0,Y 209.842,Z 472.611,A -85,B 0,C 180,E1 -21080.094,E2 -21080.094} C_VEL
LIN {X 0,Y 210.721,Z 458.076,A -85,B 0,C 180,E1 -21081.779,E2 -21081.779} C_VEL
LIN {X 0,Y 211.531,Z 442.969,A -85,B 0,C 180,E1 -21083.042,E2 -21083.042} C_VEL
LIN {X 0,Y 213.65,Z 384.472,A -85,B 0,C 180,E1 -21086.381,E2 -21086.381} C_VEL
LIN {X 0,Y 213.657,Z 380.353,A -85,B 0,C 180,E1 -21086.615,E2 -21086.615} C_VEL
LIN {X 0,Y 206.798,Z 355.723,A -85,B 0,C 180,E1 -21088.348,E2 -21088.348} C_VEL
LIN {X 0,Y 206.701,Z 355.739,A -85,B 0,C 180,E1 -21092.956,E2 -21092.956} C_VEL
LIN {X 0,Y 206.678,Z 355.735,A -85,B 0,C 180,E1 -21097.739,E2 -21097.739} C_VEL
LIN {X 0,Y 206.641,Z 355.743,A -85,B 0,C 180,E1 -21101.562,E2 -21101.562} C_VEL
LIN {X 0,Y 206.634,Z 355.742,A -85,B 0,C 180,E1 -21105.58,E2 -21105.58} C_VEL
LIN {X 0,Y 206.665,Z 355.74,A -85,B 0,C 180,E1 -21109.75,E2 -21109.75} C_VEL
LIN {X 0,Y 206.729,Z 355.731,A -85,B 0,C 180,E1 -21114.695,E2 -21114.695} C_VEL
LIN {X 0,Y 206.704,Z 355.736,A -85,B 0,C 180,E1 -21119.336,E2 -21119.336} C_VEL
LIN {X 0,Y 206.73,Z 355.729,A -85,B 0,C 180,E1 -21123.772,E2 -21123.772} C_VEL
LIN {X 0,Y 206.755,Z 355.73,A -85,B 0,C 180,E1 -21128.043,E2 -21128.043} C_VEL
LIN {X 0,Y 206.871,Z 355.714,A -85,B 0,C 180,E1 -21132.197,E2 -21132.197} C_VEL
LIN {X 0,Y 206.912,Z 355.711,A -85,B 0,C 180,E1 -21136.246,E2 -21136.246} C_VEL
LIN {X 0,Y 207.13,Z 355.683,A -85,B 0,C 180,E1 -21140.233,E2 -21140.233} C_VEL
LIN {X 0,Y 207.186,Z 355.673,A -85,B 0,C 180,E1 -21142.202,E2 -21142.202} C_VEL
LIN {X 0,Y 207.381,Z 355.652,A -85,B 0,C 180,E1 -21148.058,E2 -21148.058} C_VEL
LIN {X 0,Y 207.513,Z 355.632,A -85,B 0,C 180,E1 -21150,E2 -21150} C_VEL
LIN {X 0,Y 207.381,Z 355.65,A -85,B 0,C 180,E1 -21151.942,E2 -21151.942} C_VEL
LIN {X 0,Y 207.187,Z 355.674,A -85,B 0,C 180,E1 -21157.799,E2 -21157.799} C_VEL
LIN {X 0,Y 206.981,Z 355.701,A -85,B 0,C 180,E1 -21161.755,E2 -21161.755} C_VEL
LIN {X 0,Y 206.865,Z 355.715,A -85,B 0,C 180,E1 -21165.771,E2 -21165.771} C_VEL
LIN {X 0,Y 206.782,Z 355.726,A -85,B 0,C 180,E1 -21169.87,E2 -21169.87} C_VEL
LIN {X 0,Y 206.762,Z 355.729,A -85,B 0,C 180,E1 -21174.073,E2 -21174.073} C_VEL
LIN {X 0,Y 206.735,Z 355.733,A -85,B 0,C 180,E1 -21178.421,E2 -21178.421} C_VEL
LIN {X 0,Y 206.705,Z 355.733,A -85,B 0,C 180,E1 -21182.957,E2 -21182.957} C_VEL
LIN {X 0,Y 206.721,Z 355.731,A -85,B 0,C 180,E1 -21185.321,E2 -21185.321} C_VEL
LIN {X 0,Y 206.666,Z 355.741,A -85,B 0,C 180,E1 -21190.251,E2 -21190.251} C_VEL
LIN {X 0,Y 206.633,Z 355.744,A -85,B 0,C 180,E1 -21195.583,E2 -21195.583} C_VEL
LIN {X 0,Y 206.663,Z 355.741,A -85,B 0,C 180,E1 -21199.751,E2 -21199.751} C_VEL
LIN {X 0,Y 206.772,Z 355.727,A -85,B 0,C 180,E1 -21204.704,E2 -21204.704} C_VEL
LIN {X 0,Y 214.771,Z 382.797,A -85,B 0,C 180,E1 -21206.637,E2 -21206.637} C_VEL
LIN {X 0,Y 212.721,Z 433.277,A -85,B 0,C 180,E1 -21209.253,E2 -21209.253} C_VEL
LIN {X 0,Y 212.17,Z 448.299,A -85,B 0,C 180,E1 -21210.208,E2 -21210.208} C_VEL
LIN {X 0,Y 211.392,Z 461.813,A -85,B 0,C 180,E1 -21211.452,E2 -21211.452} C_VEL
LIN {X 0,Y 210.507,Z 474.168,A -85,B 0,C 180,E1 -21212.944,E2 -21212.944} C_VEL
LIN {X 0,Y 209.446,Z 487.158,A -85,B 0,C 180,E1 -21214.959,E2 -21214.959} C_VEL
LIN {X 0,Y 208.405,Z 498.633,A -85,B 0,C 180,E1 -21217.183,E2 -21217.183} C_VEL
LIN {X 0,Y 207.415,Z 509.049,A -85,B 0,C 180,E1 -21219.678,E2 -21219.678} C_VEL
LIN {X 0,Y 206.744,Z 517.714,A -85,B 0,C 180,E1 -21222.186,E2 -21222.186} C_VEL
LIN {X 0,Y 206.231,Z 526.169,A -85,B 0,C 180,E1 -21225.193,E2 -21225.193} C_VEL
LIN {X 0,Y 205.984,Z 532.951,A -85,B 0,C 180,E1 -21228.188,E2 -21228.188} C_VEL
LIN {X 0,Y 206.205,Z 538.576,A -85,B 0,C 180,E1 -21231.266,E2 -21231.266} C_VEL
LIN {X 0,Y 206.574,Z 542.707,A -85,B 0,C 180,E1 -21234.143,E2 -21234.143} C_VEL
LIN {X 0,Y 207.08,Z 544.955,A -85,B 0,C 180,E1 -21236.109,E2 -21236.109} C_VEL
LIN {X 0,Y 208.806,Z 548.159,A -85,B 0,C 180,E1 -21240.001,E2 -21240.001} C_VEL
LIN {X 0,Y 209.931,Z 549.128,A -85,B 0,C 180,E1 -21241.919,E2 -21241.919} C_VEL
LIN {X 0,Y 212.792,Z 549.829,A -85,B 0,C 180,E1 -21245.687,E2 -21245.687} C_VEL
LIN {X 0,Y 214.556,Z 549.588,A -85,B 0,C 180,E1 -21247.53,E2 -21247.53} C_VEL
LIN {X 0,Y 216.541,Z 548.905,A -85,B 0,C 180,E1 -21249.34,E2 -21249.34} C_VEL
LIN {X 0,Y 221.022,Z 546.345,A -85,B 0,C 180,E1 -21252.862,E2 -21252.862} C_VEL
LIN {X 0,Y 224.904,Z 543.298,A -85,B 0,C 180,E1 -21255.404,E2 -21255.404} C_VEL
LIN {X 0,Y 229.197,Z 539.198,A -85,B 0,C 180,E1 -21257.857,E2 -21257.857} C_VEL
LIN {X 0,Y 234.657,Z 532.948,A -85,B 0,C 180,E1 -21260.605,E2 -21260.605} C_VEL
LIN {X 0,Y 239.754,Z 526.195,A -85,B 0,C 180,E1 -21262.856,E2 -21262.856} C_VEL
LIN {X 0,Y 245.163,Z 517.865,A -85,B 0,C 180,E1 -21265.014,E2 -21265.014} C_VEL
LIN {X 0,Y 250.865,Z 507.605,A -85,B 0,C 180,E1 -21267.081,E2 -21267.081} C_VEL
LIN {X 0,Y 256.27,Z 495.878,A -85,B 0,C 180,E1 -21268.905,E2 -21268.905} C_VEL
LIN {X 0,Y 260.782,Z 484.088,A -85,B 0,C 180,E1 -21270.308,E2 -21270.308} C_VEL
LIN {X 0,Y 264.403,Z 472.118,A -85,B 0,C 180,E1 -21271.443,E2 -21271.443} C_VEL
LIN {X 0,Y 267.488,Z 458.807,A -85,B 0,C 180,E1 -21272.429,E2 -21272.429} C_VEL
LIN {X 0,Y 271.999,Z 434.514,A -85,B 0,C 180,E1 -21273.671,E2 -21273.671} C_VEL
LIN {X 0,Y 272.238,Z 433.141,A -85,B 0,C 180,E1 -21273.755,E2 -21273.755} C_VEL
LIN {X 0,Y 271.284,Z 430.448,A -85,B 0,C 180,E1 -21275.52,E2 -21275.52} C_VEL
LIN {X 0,Y 270.526,Z 428.44,A -85,B 0,C 180,E1 -21277.728,E2 -21277.728} C_VEL
LIN {X 0,Y 270.075,Z 428.69,A -85,B 0,C 180,E1 -21280.006,E2 -21280.006} C_VEL
LIN {X 0,Y 270.202,Z 429.858,A -85,B 0,C 180,E1 -21281.963,E2 -21281.963} C_VEL
LIN {X 0,Y 270.261,Z 431.137,A -85,B 0,C 180,E1 -21282.716,E2 -21282.716} C_VEL
LIN {X 0,Y 270.042,Z 433.523,A -85,B 0,C 180,E1 -21283.35,E2 -21283.35} C_VEL
LIN {X 0,Y 269.617,Z 436.623,A -85,B 0,C 180,E1 -21283.87,E2 -21283.87} C_VEL
LIN {X 0,Y 269.061,Z 440.091,A -85,B 0,C 180,E1 -21284.27,E2 -21284.27} C_VEL
LIN {X 0,Y 267.62,Z 448.328,A -85,B 0,C 180,E1 -21284.908,E2 -21284.908} C_VEL
LIN {X 0,Y 266.129,Z 456.669,A -85,B 0,C 180,E1 -21285.491,E2 -21285.491} C_VEL
LIN {X 0,Y 263.912,Z 470.181,A -85,B 0,C 180,E1 -21286.548,E2 -21286.548} C_VEL
LIN {X 0,Y 260.079,Z 485.888,A -85,B 0,C 180,E1 -21287.314,E2 -21287.314} C_VEL
LIN {X 0,Y 255.492,Z 499.696,A -85,B 0,C 180,E1 -21288.159,E2 -21288.159} C_VEL
LIN {X 0,Y 250.117,Z 512.937,A -85,B 0,C 180,E1 -21289.208,E2 -21289.208} C_VEL
LIN {X 0,Y 243.689,Z 526.203,A -85,B 0,C 180,E1 -21290.618,E2 -21290.618} C_VEL
LIN {X 0,Y 237.606,Z 537.081,A -85,B 0,C 180,E1 -21292.138,E2 -21292.138} C_VEL
LIN {X 0,Y 230.777,Z 547.966,A -85,B 0,C 180,E1 -21294.109,E2 -21294.109} C_VEL
LIN {X 0,Y 224.526,Z 556.961,A -85,B 0,C 180,E1 -21296.247,E2 -21296.247} C_VEL
LIN {X 0,Y 218.9,Z 564.498,A -85,B 0,C 180,E1 -21298.552,E2 -21298.552} C_VEL
LIN {X 0,Y 213.216,Z 571.699,A -85,B 0,C 180,E1 -21301.448,E2 -21301.448} C_VEL
LIN {X 0,Y 208.94,Z 576.767,A -85,B 0,C 180,E1 -21304.069,E2 -21304.069} C_VEL
LIN {X 0,Y 204.321,Z 582.048,A -85,B 0,C 180,E1 -21307.767,E2 -21307.767} C_VEL
LIN {X 0,Y 202.526,Z 584.116,A -85,B 0,C 180,E1 -21309.695,E2 -21309.695} C_VEL
LIN {X 0,Y 199.911,Z 587.107,A -85,B 0,C 180,E1 -21313.665,E2 -21313.665} C_VEL
LIN {X 0,Y 198.521,Z 588.685,A -85,B 0,C 180,E1 -21317.736,E2 -21317.736} C_VEL
LIN {X 0,Y 198.439,Z 588.845,A -85,B 0,C 180,E1 -21321.855,E2 -21321.855} C_VEL
LIN {X 0,Y 198.826,Z 588.348,A -85,B 0,C 180,E1 -21323.912,E2 -21323.912} C_VEL
LIN {X 0,Y 199.372,Z 587.454,A -85,B 0,C 180,E1 -21325.957,E2 -21325.957} C_VEL
LIN {X 0,Y 200.054,Z 586.128,A -85,B 0,C 180,E1 -21327.986,E2 -21327.986} C_VEL
LIN {X 0,Y 200.939,Z 583.722,A -85,B 0,C 180,E1 -21330.626,E2 -21330.626} C_VEL
LIN {X 0,Y 199.689,Z 586.651,A -85,B 0,C 180,E1 -21334.036,E2 -21334.036} C_VEL
LIN {X 0,Y 198.715,Z 588.498,A -85,B 0,C 180,E1 -21337.988,E2 -21337.988} C_VEL
LIN {X 0,Y 198.639,Z 588.926,A -85,B 0,C 180,E1 -21342.256,E2 -21342.256} C_VEL
LIN {X 0,Y 199.959,Z 587.942,A -85,B 0,C 180,E1 -21346.33,E2 -21346.33} C_VEL
LIN {X 0,Y 202.544,Z 585.606,A -85,B 0,C 180,E1 -21350.303,E2 -21350.303} C_VEL
LIN {X 0,Y 206.538,Z 581.934,A -85,B 0,C 180,E1 -21354.1,E2 -21354.1} C_VEL
LIN {X 0,Y 211.806,Z 576.814,A -85,B 0,C 180,E1 -21357.68,E2 -21357.68} C_VEL
LIN {X 0,Y 216.519,Z 571.95,A -85,B 0,C 180,E1 -21360.206,E2 -21360.206} C_VEL
LIN {X 0,Y 223.821,Z 563.915,A -85,B 0,C 180,E1 -21363.333,E2 -21363.333} C_VEL
LIN {X 0,Y 231.021,Z 555.286,A -85,B 0,C 180,E1 -21365.846,E2 -21365.846} C_VEL
LIN {X 0,Y 237.903,Z 546.391,A -85,B 0,C 180,E1 -21367.806,E2 -21367.806} C_VEL
LIN {X 0,Y 245.313,Z 535.76,A -85,B 0,C 180,E1 -21369.601,E2 -21369.601} C_VEL
LIN {X 0,Y 253.037,Z 523.234,A -85,B 0,C 180,E1 -21371.232,E2 -21371.232} C_VEL
LIN {X 0,Y 259.469,Z 511.378,A -85,B 0,C 180,E1 -21372.358,E2 -21372.358} C_VEL
LIN {X 0,Y 265.99,Z 497.286,A -85,B 0,C 180,E1 -21373.391,E2 -21373.391} C_VEL
LIN {X 0,Y 271.856,Z 481.63,A -85,B 0,C 180,E1 -21374.267,E2 -21374.267} C_VEL
LIN {X 0,Y 275.292,Z 469.892,A -85,B 0,C 180,E1 -21374.868,E2 -21374.868} C_VEL
LIN {X 0,Y 277.344,Z 460.891,A -85,B 0,C 180,E1 -21375.723,E2 -21375.723} C_VEL
LIN {X 0,Y 277.748,Z 458.978,A -85,B 0,C 180,E1 -21375.977,E2 -21375.977} C_VEL
LIN {X 0,Y 278.025,Z 457.227,A -85,B 0,C 180,E1 -21376.863,E2 -21376.863} C_VEL
LIN {X 0,Y 278.623,Z 455.344,A -85,B 0,C 180,E1 -21378.655,E2 -21378.655} C_VEL
LIN {X 0,Y 278.67,Z 455.249,A -85,B 0,C 180,E1 -21378.752,E2 -21378.752} C_VEL
LIN {X 0,Y 275.012,Z 469.302,A -85,B 0,C 180,E1 -21379.583,E2 -21379.583} C_VEL
LIN {X 0,Y 270.946,Z 481.417,A -85,B 0,C 180,E1 -21380.542,E2 -21380.542} C_VEL
LIN {X 0,Y 266.27,Z 492.661,A -85,B 0,C 180,E1 -21381.664,E2 -21381.664} C_VEL
LIN {X 0,Y 260.477,Z 504.189,A -85,B 0,C 180,E1 -21383.105,E2 -21383.105} C_VEL
LIN {X 0,Y 253.773,Z 515.348,A -85,B 0,C 180,E1 -21384.924,E2 -21384.924} C_VEL
LIN {X 0,Y 247.257,Z 524.476,A -85,B 0,C 180,E1 -21386.827,E2 -21386.827} C_VEL
LIN {X 0,Y 241.062,Z 531.992,A -85,B 0,C 180,E1 -21388.835,E2 -21388.835} C_VEL
LIN {X 0,Y 234.288,Z 538.983,A -85,B 0,C 180,E1 -21391.317,E2 -21391.317} C_VEL
LIN {X 0,Y 228.847,Z 543.742,A -85,B 0,C 180,E1 -21393.556,E2 -21393.556} C_VEL
LIN {X 0,Y 223.814,Z 547.456,A -85,B 0,C 180,E1 -21395.906,E2 -21395.906} C_VEL
LIN {X 0,Y 219.762,Z 549.924,A -85,B 0,C 180,E1 -21398.036,E2 -21398.036} C_VEL
LIN {X 0,Y 214.998,Z 552.051,A -85,B 0,C 180,E1 -21400.919,E2 -21400.919} C_VEL
LIN {X 0,Y 210.049,Z 553.137,A -85,B 0,C 180,E1 -21404.473,E2 -21404.473} C_VEL
LIN {X 0,Y 207.96,Z 553.102,A -85,B 0,C 180,E1 -21406.315,E2 -21406.315} C_VEL
LIN {X 0,Y 206.031,Z 552.668,A -85,B 0,C 180,E1 -21408.189,E2 -21408.189} C_VEL
LIN {X 0,Y 202.989,Z 550.605,A -85,B 0,C 180,E1 -21412.039,E2 -21412.039} C_VEL
LIN {X 0,Y 201.237,Z 548.032,A -85,B 0,C 180,E1 -21414.99,E2 -21414.99} C_VEL
LIN {X 0,Y 199.976,Z 544.521,A -85,B 0,C 180,E1 -21417.985,E2 -21417.985} C_VEL
LIN {X 0,Y 199.13,Z 539.996,A -85,B 0,C 180,E1 -21421.01,E2 -21421.01} C_VEL
LIN {X 0,Y 198.798,Z 533.308,A -85,B 0,C 180,E1 -21424.561,E2 -21424.561} C_VEL
LIN {X 0,Y 198.992,Z 527.255,A -85,B 0,C 180,E1 -21427.174,E2 -21427.174} C_VEL
LIN {X 0,Y 199.393,Z 519.017,A -85,B 0,C 180,E1 -21430.15,E2 -21430.15} C_VEL
LIN {X 0,Y 200.02,Z 508.574,A -85,B 0,C 180,E1 -21433.201,E2 -21433.201} C_VEL
LIN {X 0,Y 200.876,Z 497.996,A -85,B 0,C 180,E1 -21435.732,E2 -21435.732} C_VEL
LIN {X 0,Y 201.807,Z 484.839,A -85,B 0,C 180,E1 -21438.265,E2 -21438.265} C_VEL
LIN {X 0,Y 202.839,Z 471.518,A -85,B 0,C 180,E1 -21440.271,E2 -21440.271} C_VEL
LIN {X 0,Y 203.638,Z 457.923,A -85,B 0,C 180,E1 -21441.863,E2 -21441.863} C_VEL
LIN {X 0,Y 204.464,Z 442.919,A -85,B 0,C 180,E1 -21443.149,E2 -21443.149} C_VEL
LIN {X 0,Y 206.618,Z 384.291,A -85,B 0,C 180,E1 -21446.631,E2 -21446.631} C_VEL
LIN {X 0,Y 206.638,Z 381.52,A -85,B 0,C 180,E1 -21446.795,E2 -21446.795} C_VEL
LIN {X 0,Y 199.77,Z 356.6,A -85,B 0,C 180,E1 -21448.6,E2 -21448.6} C_VEL
LIN {X 0,Y 199.677,Z 356.61,A -85,B 0,C 180,E1 -21452.357,E2 -21452.357} C_VEL
LIN {X 0,Y 199.621,Z 356.618,A -85,B 0,C 180,E1 -21456.762,E2 -21456.762} C_VEL
LIN {X 0,Y 199.607,Z 356.618,A -85,B 0,C 180,E1 -21459.327,E2 -21459.327} C_VEL
LIN {X 0,Y 199.573,Z 356.624,A -85,B 0,C 180,E1 -21462.31,E2 -21462.31} C_VEL
LIN {X 0,Y 199.58,Z 356.622,A -85,B 0,C 180,E1 -21465.229,E2 -21465.229} C_VEL
LIN {X 0,Y 199.637,Z 356.619,A -85,B 0,C 180,E1 -21470.679,E2 -21470.679} C_VEL
LIN {X 0,Y 199.63,Z 356.612,A -85,B 0,C 180,E1 -21475.717,E2 -21475.717} C_VEL
LIN {X 0,Y 199.694,Z 356.608,A -85,B 0,C 180,E1 -21478.136,E2 -21478.136} C_VEL
LIN {X 0,Y 199.683,Z 356.609,A -85,B 0,C 180,E1 -21482.771,E2 -21482.771} C_VEL
LIN {X 0,Y 199.736,Z 356.604,A -85,B 0,C 180,E1 -21487.229,E2 -21487.229} C_VEL
LIN {X 0,Y 199.794,Z 356.594,A -85,B 0,C 180,E1 -21491.757,E2 -21491.757} C_VEL
LIN {X 0,Y 199.846,Z 356.589,A -85,B 0,C 180,E1 -21495.749,E2 -21495.749} C_VEL
LIN {X 0,Y 200.073,Z 356.56,A -85,B 0,C 180,E1 -21499.885,E2 -21499.885} C_VEL
